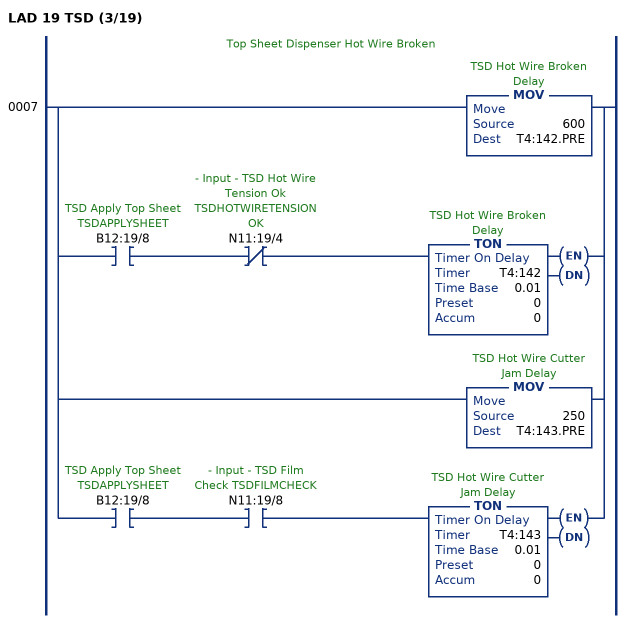
% Rung: 7 %
% Top Sheet Dispenser Hot Wire Broken %
SOR BST MOV 600 T4:142.PRE NXB XIC B12:19/8 XIO N11:19/4 TON T4:142 0.01 0 0 NXB MOV 250 T4:143.PRE NXB XIC B12:19/8 XIC N11:19/8 TON T4:143 0.01 0 0 BND EOR
%   T4:142  "TSD Hot Wire Broken Delay" %
%   B12:19/8  TSDAPPLYSHEET  "TSD Apply Top Sheet" %
%   N11:19/4  TSDHOTWIRETENSIONOK  "- Input - TSD Hot Wire Tension Ok" %
%   T4:143  "TSD Hot Wire Cutter Jam Delay" %
%   N11:19/8  TSDFILMCHECK  "- Input - TSD Film Check" %

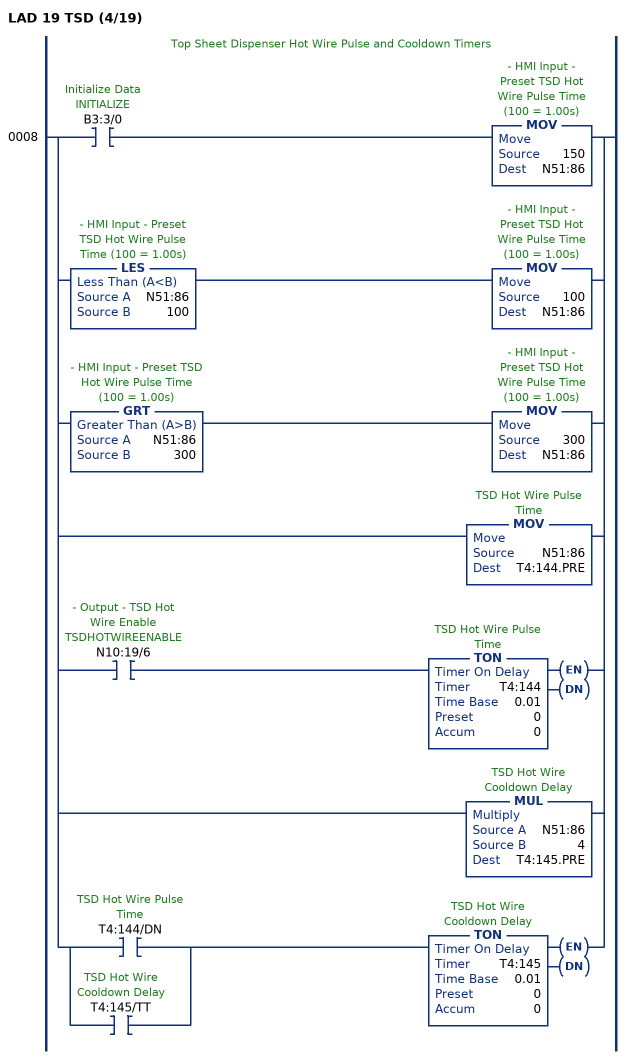
% Rung: 8 %
% Top Sheet Dispenser Hot Wire Pulse and Cooldown Timers %
SOR BST BST XIC B3:3/0 MOV 150 N51:86 NXB LES N51:86 100 MOV 100 N51:86 NXB GRT N51:86 300 MOV 300 N51:86 NXB MOV N51:86 T4:144.PRE BND NXB XIC N10:19/6 TON T4:144 0.01 0 0 NXB MUL N51:86 4 T4:145.PRE NXB BST XIC T4:144/DN NXB XIC T4:145/TT BND TON T4:145 0.01 0 0 BND EOR
%   B3:3/0  INITIALIZE  "Initialize Data" %
%   N51:86  "- HMI Input - Preset TSD Hot Wire Pulse Time (100 = 1.00s)" %
%   T4:144  "TSD Hot Wire Pulse Time" %
%   N10:19/6  TSDHOTWIREENABLE  "- Output - TSD Hot Wire Enable" %
%   T4:145  "TSD Hot Wire Cooldown Delay" %

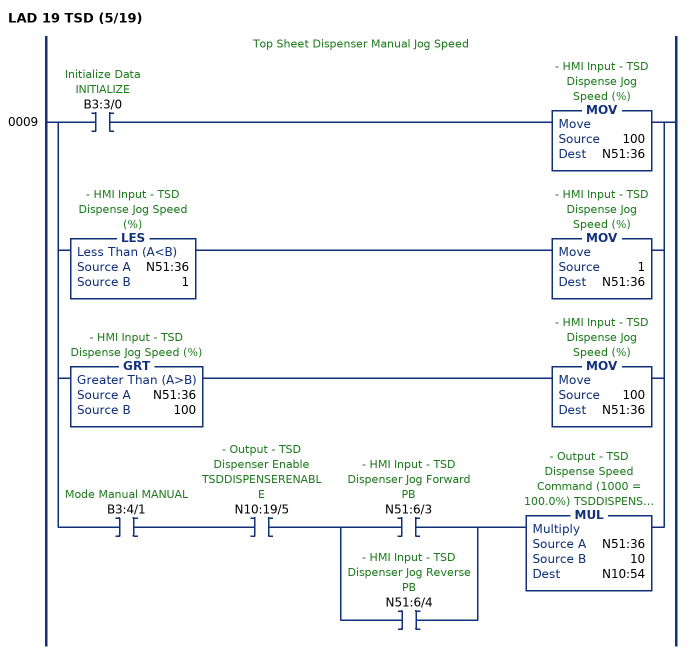
% Rung: 9 %
% Top Sheet Dispenser Manual Jog Speed %
SOR BST XIC B3:3/0 MOV 100 N51:36 NXB LES N51:36 1 MOV 1 N51:36 NXB GRT N51:36 100 MOV 100 N51:36 NXB XIC B3:4/1 XIC N10:19/5 BST XIC N51:6/3 NXB XIC N51:6/4 BND MUL N51:36 10 N10:54 BND EOR
%   B3:3/0  INITIALIZE  "Initialize Data" %
%   N51:36  "- HMI Input - TSD Dispense Jog Speed (%)" %
%   B3:4/1  MANUAL  "Mode Manual" %
%   N10:19/5  TSDDISPENSERENABLE  "- Output - TSD Dispenser Enable" %
%   N51:6/3  "- HMI Input - TSD Dispenser Jog Forward PB" %
%   N51:6/4  "- HMI Input - TSD Dispenser Jog Reverse PB" %
%   N10:54  TSDDISPENSECOMMAND  "- Output - TSD Dispense Speed Command (1000 = 100.0%)" %

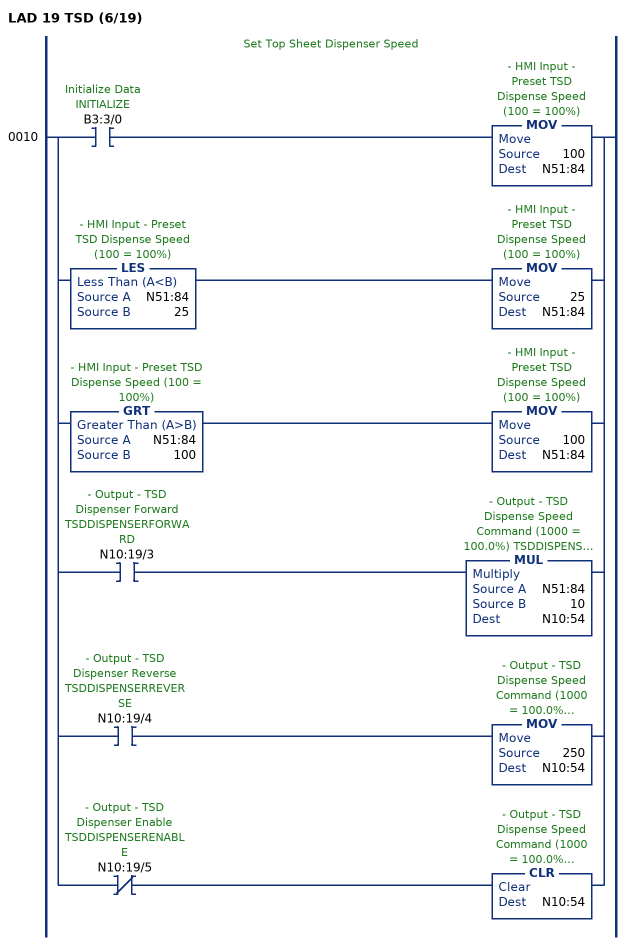
% Rung: 10 %
% Set Top Sheet Dispenser Speed %
SOR BST BST XIC B3:3/0 MOV 100 N51:84 NXB LES N51:84 25 MOV 25 N51:84 NXB GRT N51:84 100 MOV 100 N51:84 BND NXB XIC N10:19/3 MUL N51:84 10 N10:54 NXB XIC N10:19/4 MOV 250 N10:54 NXB XIO N10:19/5 CLR N10:54 BND EOR
%   B3:3/0  INITIALIZE  "Initialize Data" %
%   N51:84  "- HMI Input - Preset TSD Dispense Speed (100 = 100%)" %
%   N10:19/3  TSDDISPENSERFORWARD  "- Output - TSD Dispenser Forward" %
%   N10:54  TSDDISPENSECOMMAND  "- Output - TSD Dispense Speed Command (1000 = 100.0%)" %
%   N10:19/4  TSDDISPENSERREVERSE  "- Output - TSD Dispenser Reverse" %
%   N10:19/5  TSDDISPENSERENABLE  "- Output - TSD Dispenser Enable" %

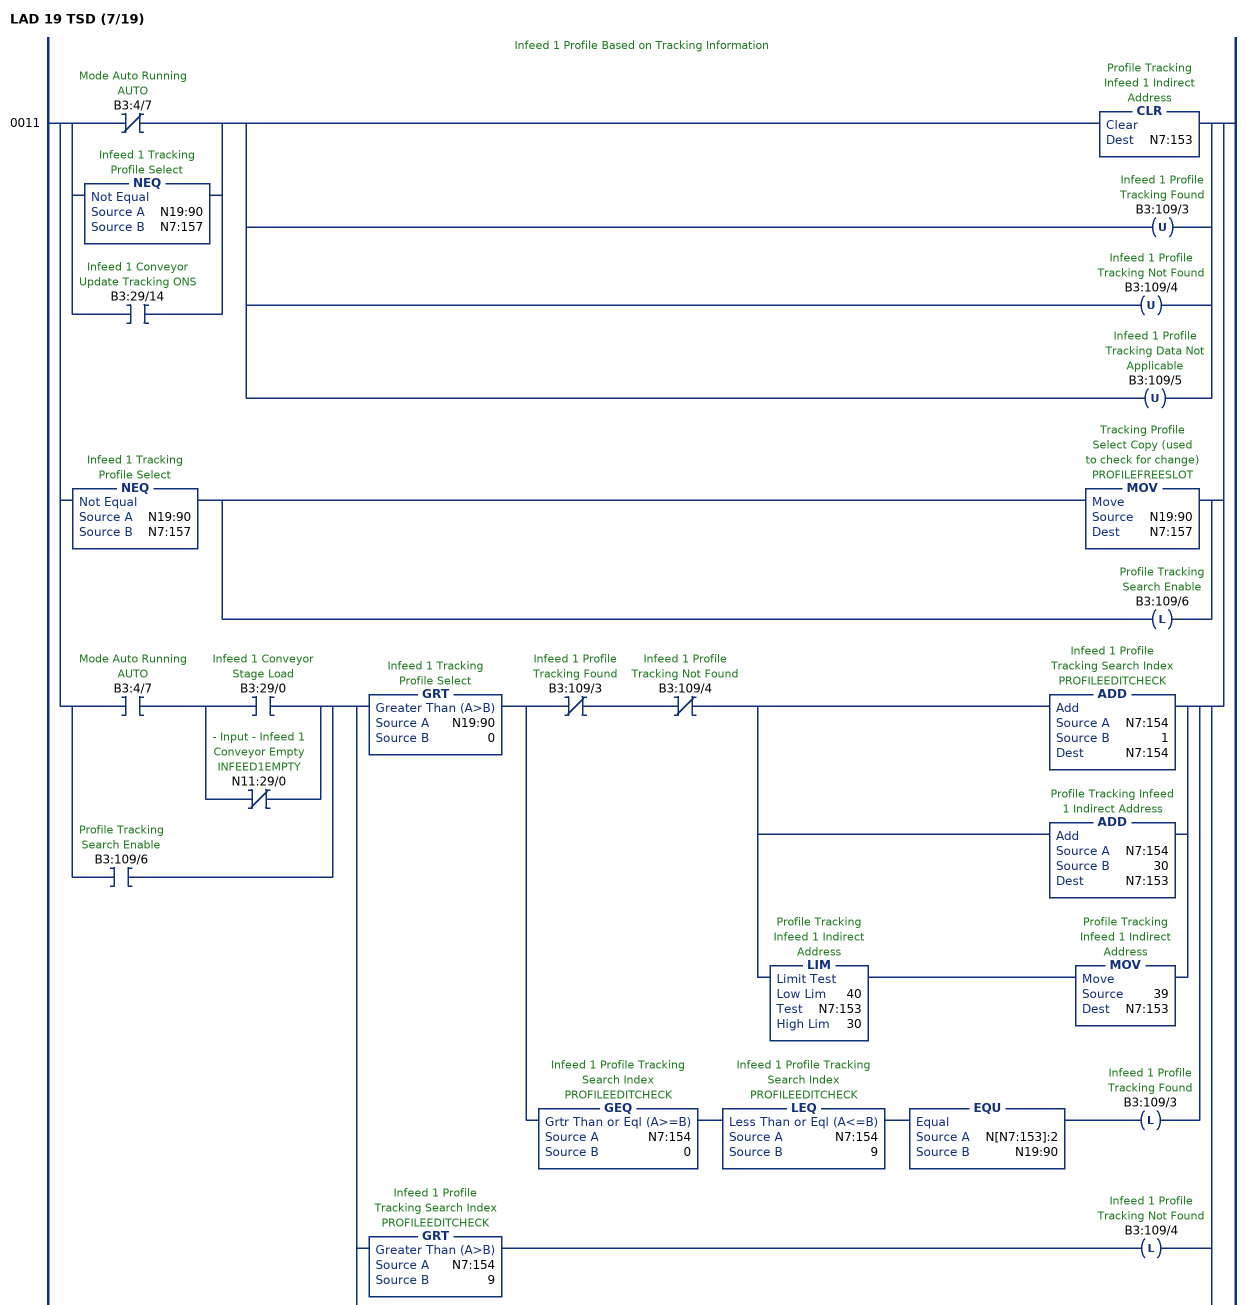

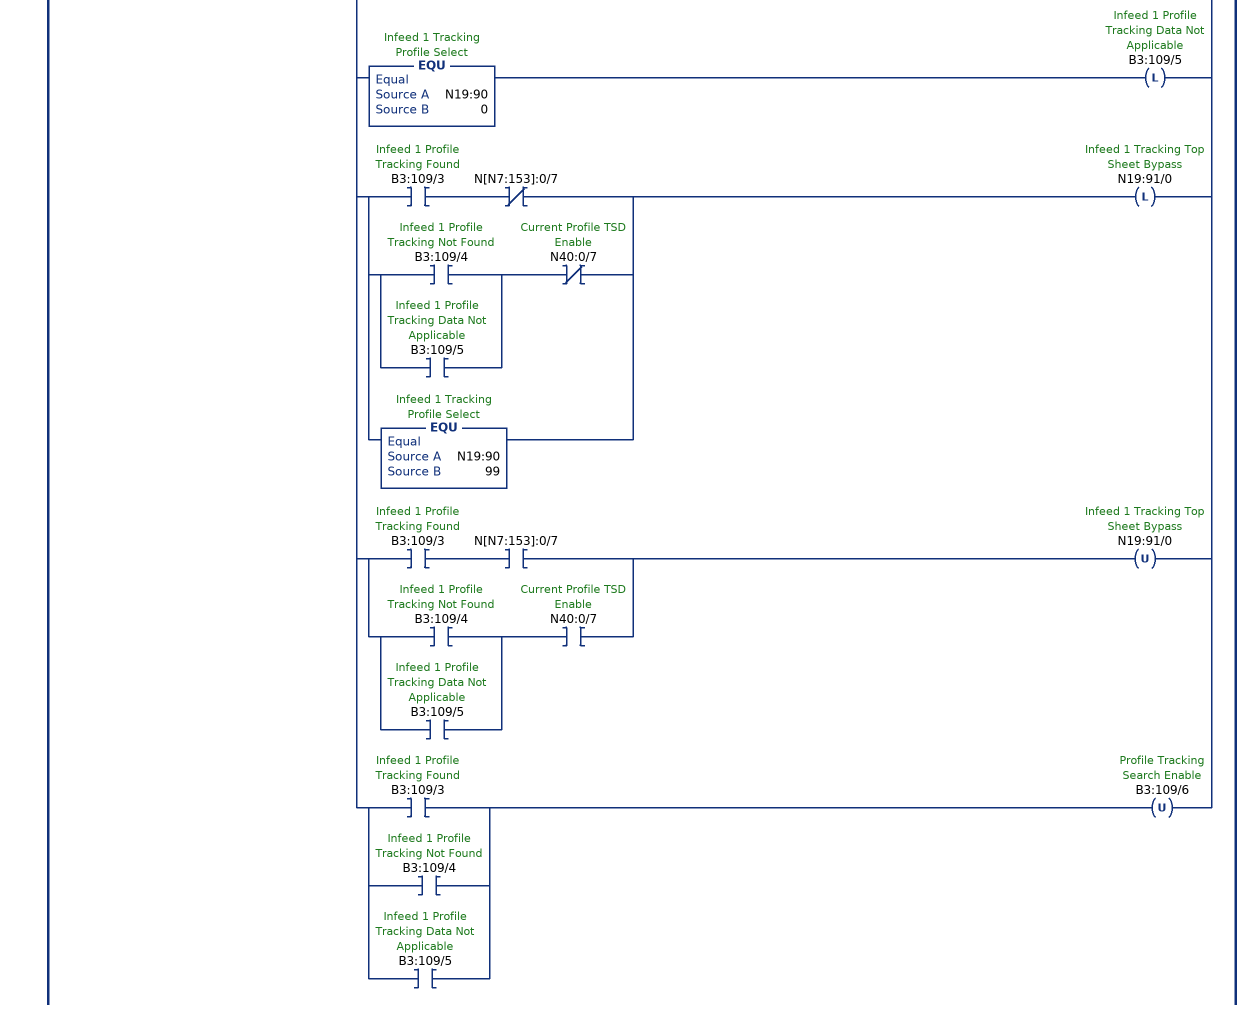
% Rung: 11 %
% Infeed 1 Profile Based on Tracking Information %
SOR BST BST XIO B3:4/7 NXB NEQ N19:90 N7:157 NXB XIC B3:29/14 BND BST CLR N7:153 NXB OTU B3:109/3 NXB OTU B3:109/4 NXB OTU B3:109/5 BND NXB NEQ N19:90 N7:157 BST MOV N19:90 N7:157 NXB OTL B3:109/6 BND NXB BST XIC B3:4/7 BST XIC B3:29/0 NXB XIO N11:29/0 BND NXB XIC B3:109/6 BND BST GRT N19:90 0 BST XIO B3:109/3 XIO B3:109/4 BST ADD N7:154 1 N7:154 NXB ADD N7:154 30 N7:153 NXB LIM 40 N7:153 30 MOV 39 N7:153 BND NXB GEQ N7:154 0 LEQ N7:154 9 EQU N[N7:153]:2 N19:90 OTL B3:109/3 BND NXB GRT N7:154 9 OTL B3:109/4 NXB EQU N19:90 0 OTL B3:109/5 NXB BST XIC B3:109/3 XIO N[N7:153]:0/7 NXB BST XIC B3:109/4 NXB XIC B3:109/5 BND XIO N40:0/7 NXB EQU N19:90 99 BND OTL N19:91/0 NXB BST XIC B3:109/3 XIC N[N7:153]:0/7 NXB BST XIC B3:109/4 NXB XIC B3:109/5 BND XIC N40:0/7 BND OTU N19:91/0 NXB BST XIC B3:109/3 NXB XIC B3:109/4 NXB XIC B3:109/5 BND OTU B3:109/6 BND BND EOR
%   B3:4/7  AUTO  "Mode Auto Running" %
%   N19:90  "Infeed 1 Tracking Profile Select" %
%   N7:157  PROFILEFREESLOT  "Tracking Profile Select Copy (used to check for change)" %
%   B3:29/14  "Infeed 1 Conveyor Update Tracking ONS" %
%   N7:153  "Profile Tracking Infeed 1 Indirect Address" %
%   B3:109/3  "Infeed 1 Profile Tracking Found" %
%   B3:109/4  "Infeed 1 Profile Tracking Not Found" %
%   B3:109/5  "Infeed 1 Profile Tracking Data Not Applicable" %
%   B3:109/6  "Profile Tracking Search Enable" %
%   B3:29/0  "Infeed 1 Conveyor Stage Load" %
%   N11:29/0  INFEED1EMPTY  "- Input - Infeed 1 Conveyor Empty" %
%   N7:154  PROFILEEDITCHECK  "Infeed 1 Profile Tracking Search Index" %
%   N40:0/7  "Current Profile TSD Enable" %
%   N19:91/0  "Infeed 1 Tracking Top Sheet Bypass" %

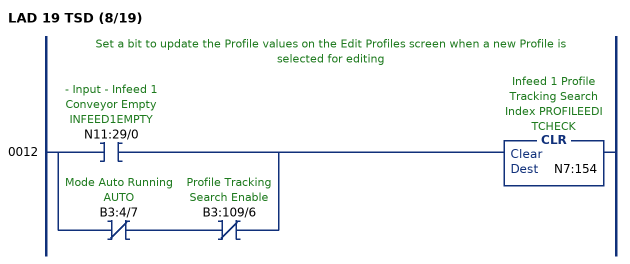
% Rung: 12 %
% Set a bit to update the Profile values on the Edit Profiles screen when a new Profile is selected for editing %
SOR BST XIC N11:29/0 NXB XIO B3:4/7 XIO B3:109/6 BND CLR N7:154 EOR
%   N11:29/0  INFEED1EMPTY  "- Input - Infeed 1 Conveyor Empty" %
%   B3:4/7  AUTO  "Mode Auto Running" %
%   B3:109/6  "Profile Tracking Search Enable" %
%   N7:154  PROFILEEDITCHECK  "Infeed 1 Profile Tracking Search Index" %

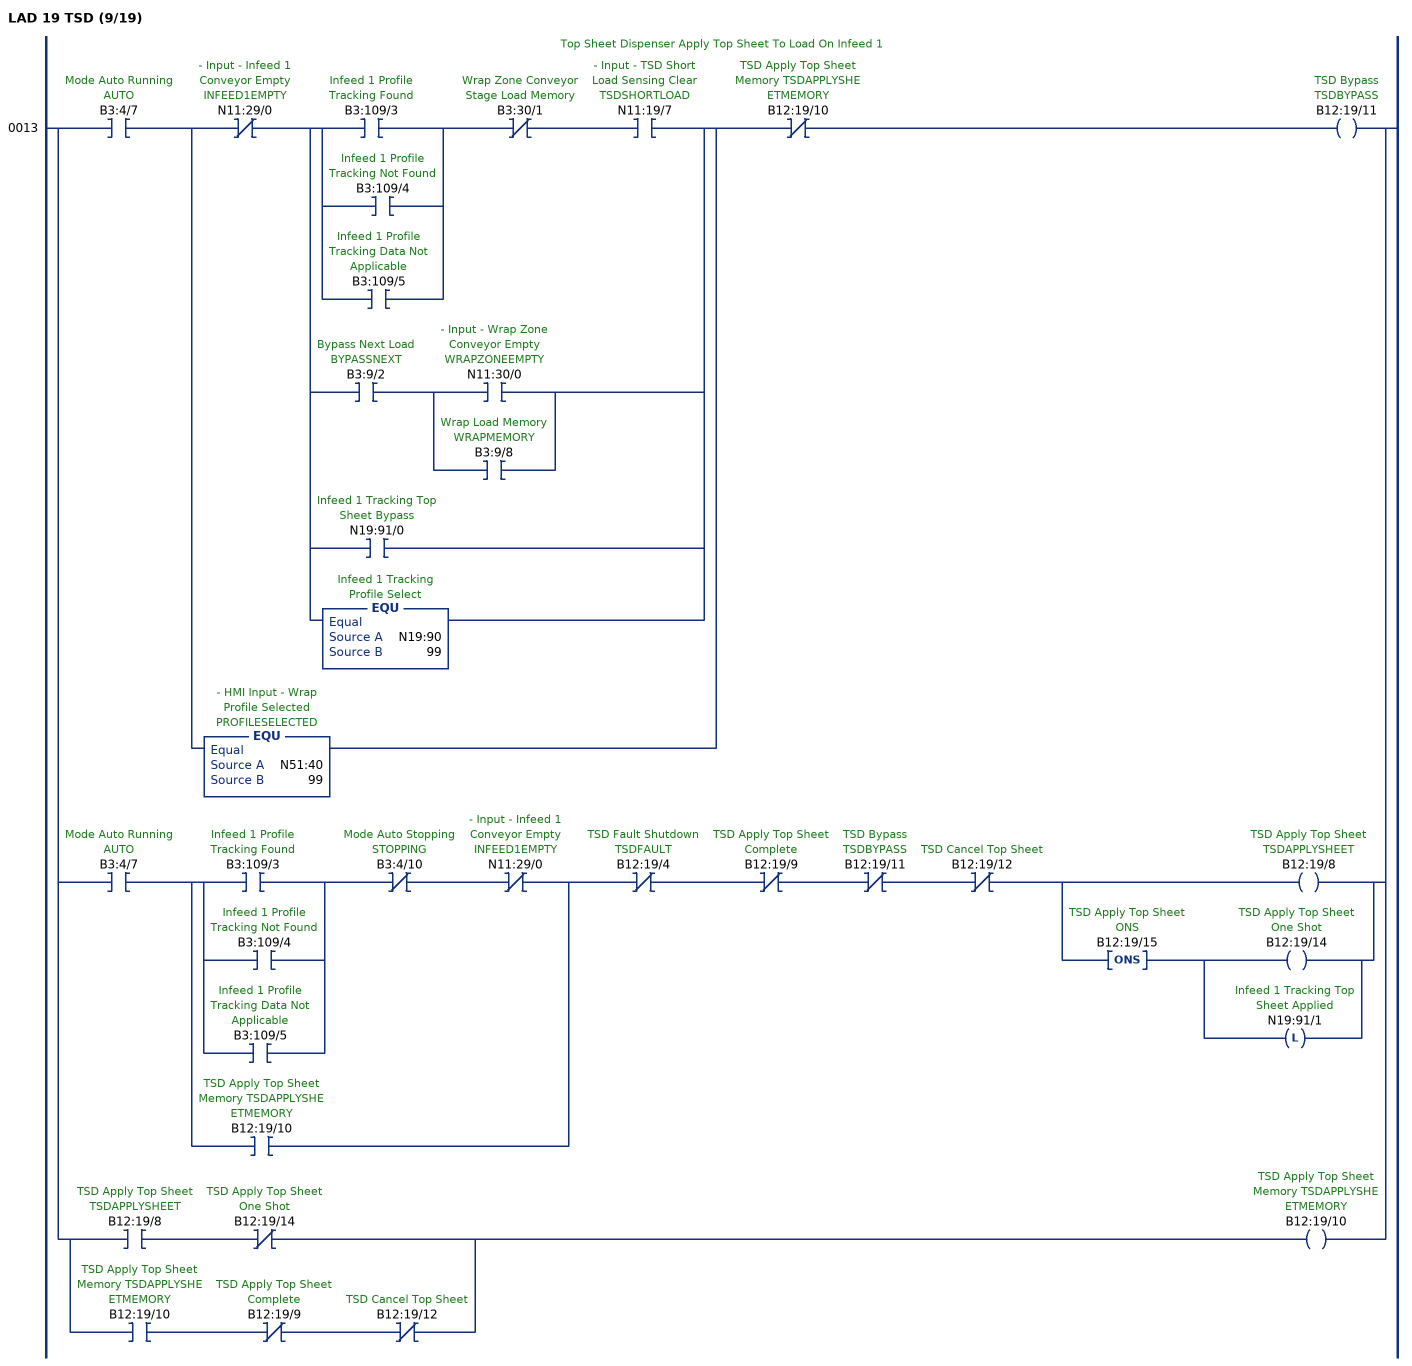
% Rung: 13 %
% Top Sheet Dispenser Apply Top Sheet To Load On Infeed 1 %
SOR BST XIC B3:4/7 BST XIO N11:29/0 BST BST XIC B3:109/3 NXB XIC B3:109/4 NXB XIC B3:109/5 BND XIO B3:30/1 XIC N11:19/7 NXB XIC B3:9/2 BST XIC N11:30/0 NXB XIC B3:9/8 BND NXB XIC N19:91/0 NXB EQU N19:90 99 BND NXB EQU N51:40 99 BND XIO B12:19/10 OTE B12:19/11 NXB XIC B3:4/7 BST BST XIC B3:109/3 NXB XIC B3:109/4 NXB XIC B3:109/5 BND XIO B3:4/10 XIO N11:29/0 NXB XIC B12:19/10 BND XIO B12:19/4 XIO B12:19/9 XIO B12:19/11 XIO B12:19/12 BST OTE B12:19/8 NXB ONS B12:19/15 BST OTE B12:19/14 NXB OTL N19:91/1 BND BND NXB BST XIC B12:19/8 XIO B12:19/14 NXB XIC B12:19/10 XIO B12:19/9 XIO B12:19/12 BND OTE B12:19/10 BND EOR
%   B3:4/7  AUTO  "Mode Auto Running" %
%   N11:29/0  INFEED1EMPTY  "- Input - Infeed 1 Conveyor Empty" %
%   B3:109/3  "Infeed 1 Profile Tracking Found" %
%   B3:109/4  "Infeed 1 Profile Tracking Not Found" %
%   B3:109/5  "Infeed 1 Profile Tracking Data Not Applicable" %
%   B3:30/1  "Wrap Zone Conveyor Stage Load Memory" %
%   N11:19/7  TSDSHORTLOAD  "- Input - TSD Short Load Sensing Clear" %
%   B3:9/2  BYPASSNEXT  "Bypass Next Load" %
%   N11:30/0  WRAPZONEEMPTY  "- Input - Wrap Zone Conveyor Empty" %
%   B3:9/8  WRAPMEMORY  "Wrap Load Memory" %
%   N19:91/0  "Infeed 1 Tracking Top Sheet Bypass" %
%   N19:90  "Infeed 1 Tracking Profile Select" %
%   N51:40  PROFILESELECTED  "- HMI Input - Wrap Profile Selected" %
%   B12:19/10  TSDAPPLYSHEETMEMORY  "TSD Apply Top Sheet Memory" %
%   B12:19/11  TSDBYPASS  "TSD Bypass" %
%   B3:4/10  STOPPING  "Mode Auto Stopping" %
%   B12:19/4  TSDFAULT  "TSD Fault Shutdown" %
%   B12:19/9  "TSD Apply Top Sheet Complete" %
%   B12:19/12  "TSD Cancel Top Sheet" %
%   B12:19/8  TSDAPPLYSHEET  "TSD Apply Top Sheet" %
%   B12:19/15  "TSD Apply Top Sheet ONS" %
%   B12:19/14  "TSD Apply Top Sheet One Shot" %
%   N19:91/1  "Infeed 1 Tracking Top Sheet Applied" %

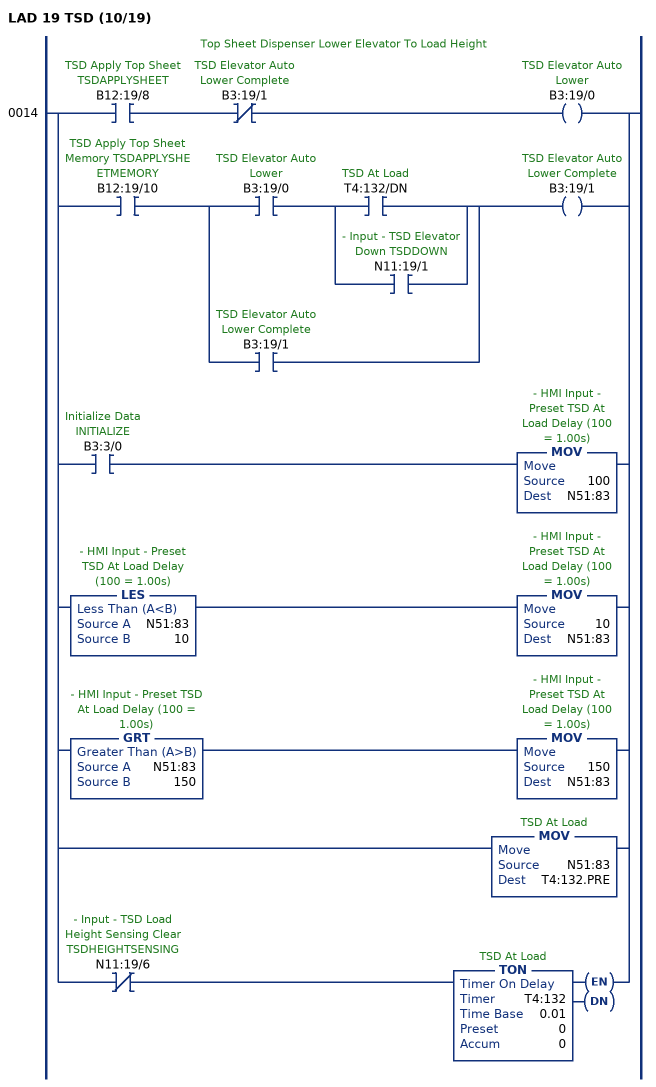
% Rung: 14 %
% Top Sheet Dispenser Lower Elevator To Load Height %
SOR BST XIC B12:19/8 XIO B3:19/1 OTE B3:19/0 NXB XIC B12:19/10 BST XIC B3:19/0 BST XIC T4:132/DN NXB XIC N11:19/1 BND NXB XIC B3:19/1 BND OTE B3:19/1 NXB BST XIC B3:3/0 MOV 100 N51:83 NXB LES N51:83 10 MOV 10 N51:83 NXB GRT N51:83 150 MOV 150 N51:83 NXB MOV N51:83 T4:132.PRE BND NXB XIO N11:19/6 TON T4:132 0.01 0 0 BND EOR
%   B12:19/8  TSDAPPLYSHEET  "TSD Apply Top Sheet" %
%   B3:19/1  "TSD Elevator Auto Lower Complete" %
%   B3:19/0  "TSD Elevator Auto Lower" %
%   B12:19/10  TSDAPPLYSHEETMEMORY  "TSD Apply Top Sheet Memory" %
%   T4:132  "TSD At Load" %
%   N11:19/1  TSDDOWN  "- Input - TSD Elevator Down" %
%   B3:3/0  INITIALIZE  "Initialize Data" %
%   N51:83  "- HMI Input - Preset TSD At Load Delay (100 = 1.00s)" %
%   N11:19/6  TSDHEIGHTSENSING  "- Input - TSD Load Height Sensing Clear" %

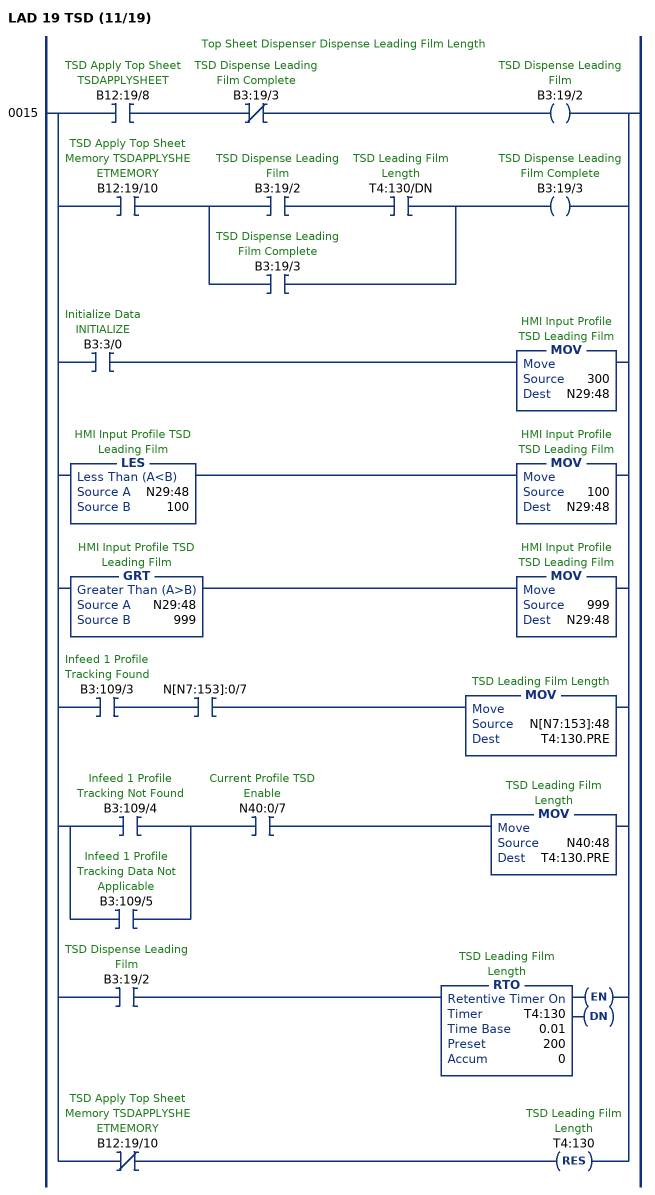
% Rung: 15 %
% Top Sheet Dispenser Dispense Leading Film Length %
SOR BST XIC B12:19/8 XIO B3:19/3 OTE B3:19/2 NXB XIC B12:19/10 BST XIC B3:19/2 XIC T4:130/DN NXB XIC B3:19/3 BND OTE B3:19/3 NXB BST XIC B3:3/0 MOV 300 N29:48 NXB LES N29:48 100 MOV 100 N29:48 NXB GRT N29:48 999 MOV 999 N29:48 NXB XIC B3:109/3 XIC N[N7:153]:0/7 MOV N[N7:153]:48 T4:130.PRE NXB BST XIC B3:109/4 NXB XIC B3:109/5 BND XIC N40:0/7 MOV N40:48 T4:130.PRE BND NXB XIC B3:19/2 RTO T4:130 0.01 200 0 NXB XIO B12:19/10 RES T4:130 BND EOR
%   B12:19/8  TSDAPPLYSHEET  "TSD Apply Top Sheet" %
%   B3:19/3  "TSD Dispense Leading Film Complete" %
%   B3:19/2  "TSD Dispense Leading Film" %
%   B12:19/10  TSDAPPLYSHEETMEMORY  "TSD Apply Top Sheet Memory" %
%   T4:130  "TSD Leading Film Length" %
%   B3:3/0  INITIALIZE  "Initialize Data" %
%   N29:48  "HMI Input Profile TSD Leading Film" %
%   B3:109/3  "Infeed 1 Profile Tracking Found" %
%   N7:153  "Profile Tracking Infeed 1 Indirect Address" %
%   B3:109/4  "Infeed 1 Profile Tracking Not Found" %
%   B3:109/5  "Infeed 1 Profile Tracking Data Not Applicable" %
%   N40:0/7  "Current Profile TSD Enable" %
%   N40:48  "Current Profile TSD Leading Film" %

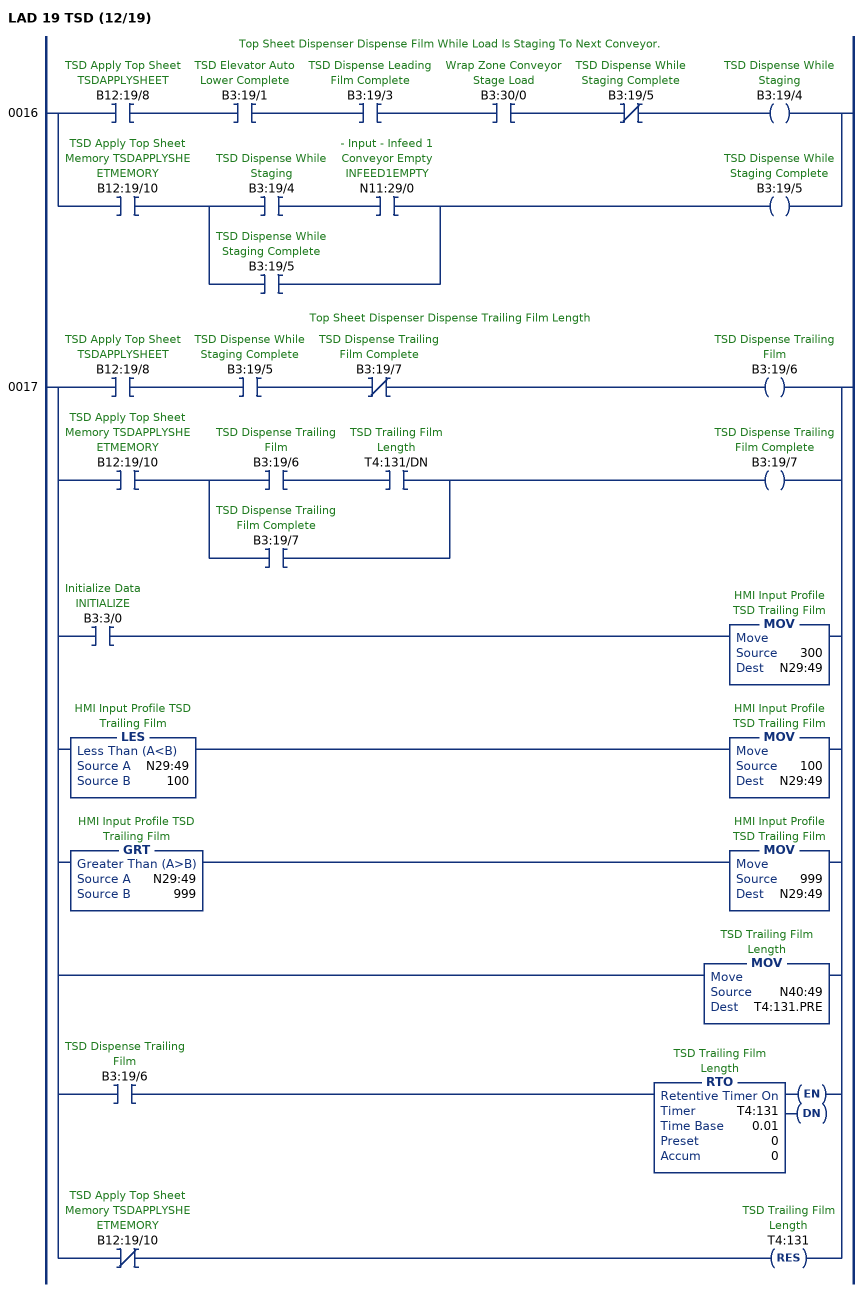
% Rung: 16 %
% Top Sheet Dispenser Dispense Film While Load Is Staging To Next Conveyor. %
SOR BST XIC B12:19/8 XIC B3:19/1 XIC B3:19/3 XIC B3:30/0 XIO B3:19/5 OTE B3:19/4 NXB XIC B12:19/10 BST XIC B3:19/4 XIC N11:29/0 NXB XIC B3:19/5 BND OTE B3:19/5 BND EOR
%   B12:19/8  TSDAPPLYSHEET  "TSD Apply Top Sheet" %
%   B3:19/1  "TSD Elevator Auto Lower Complete" %
%   B3:19/3  "TSD Dispense Leading Film Complete" %
%   B3:30/0  "Wrap Zone Conveyor Stage Load" %
%   B3:19/5  "TSD Dispense While Staging Complete" %
%   B3:19/4  "TSD Dispense While Staging" %
%   B12:19/10  TSDAPPLYSHEETMEMORY  "TSD Apply Top Sheet Memory" %
%   N11:29/0  INFEED1EMPTY  "- Input - Infeed 1 Conveyor Empty" %
% Rung: 17 %
% Top Sheet Dispenser Dispense Trailing Film Length %
SOR BST XIC B12:19/8 XIC B3:19/5 XIO B3:19/7 OTE B3:19/6 NXB XIC B12:19/10 BST XIC B3:19/6 XIC T4:131/DN NXB XIC B3:19/7 BND OTE B3:19/7 NXB BST XIC B3:3/0 MOV 300 N29:49 NXB LES N29:49 100 MOV 100 N29:49 NXB GRT N29:49 999 MOV 999 N29:49 NXB MOV N40:49 T4:131.PRE BND NXB XIC B3:19/6 RTO T4:131 0.01 0 0 NXB XIO B12:19/10 RES T4:131 BND EOR
%   B12:19/8  TSDAPPLYSHEET  "TSD Apply Top Sheet" %
%   B3:19/5  "TSD Dispense While Staging Complete" %
%   B3:19/7  "TSD Dispense Trailing Film Complete" %
%   B3:19/6  "TSD Dispense Trailing Film" %
%   B12:19/10  TSDAPPLYSHEETMEMORY  "TSD Apply Top Sheet Memory" %
%   T4:131  "TSD Trailing Film Length" %
%   B3:3/0  INITIALIZE  "Initialize Data" %
%   N29:49  "HMI Input Profile TSD Trailing Film" %
%   N40:49  "Current Profile TSD Trailing Film" %

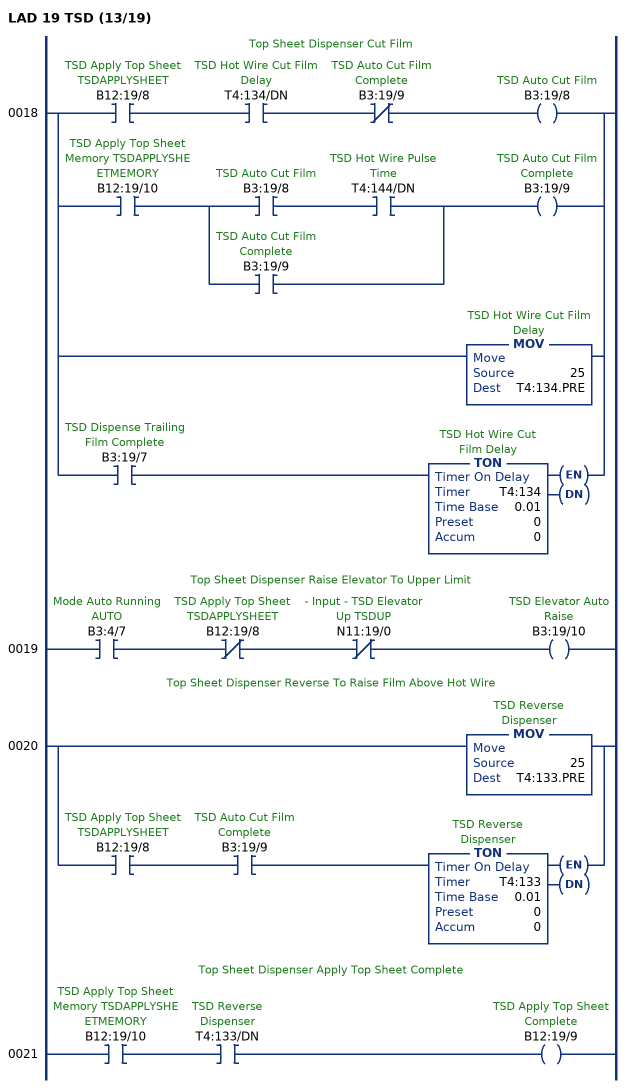
% Rung: 18 %
% Top Sheet Dispenser Cut Film %
SOR BST XIC B12:19/8 XIC T4:134/DN XIO B3:19/9 OTE B3:19/8 NXB XIC B12:19/10 BST XIC B3:19/8 XIC T4:144/DN NXB XIC B3:19/9 BND OTE B3:19/9 NXB MOV 25 T4:134.PRE NXB XIC B3:19/7 TON T4:134 0.01 0 0 BND EOR
%   B12:19/8  TSDAPPLYSHEET  "TSD Apply Top Sheet" %
%   T4:134  "TSD Hot Wire Cut Film Delay" %
%   B3:19/9  "TSD Auto Cut Film Complete" %
%   B3:19/8  "TSD Auto Cut Film" %
%   B12:19/10  TSDAPPLYSHEETMEMORY  "TSD Apply Top Sheet Memory" %
%   T4:144  "TSD Hot Wire Pulse Time" %
%   B3:19/7  "TSD Dispense Trailing Film Complete" %
% Rung: 19 %
% Top Sheet Dispenser Raise Elevator To Upper Limit %
SOR XIC B3:4/7 XIO B12:19/8 XIO N11:19/0 OTE B3:19/10 EOR
%   B3:4/7  AUTO  "Mode Auto Running" %
%   B12:19/8  TSDAPPLYSHEET  "TSD Apply Top Sheet" %
%   N11:19/0  TSDUP  "- Input - TSD Elevator Up" %
%   B3:19/10  "TSD Elevator Auto Raise" %
% Rung: 20 %
% Top Sheet Dispenser Reverse To Raise Film Above Hot Wire %
SOR BST MOV 25 T4:133.PRE NXB XIC B12:19/8 XIC B3:19/9 TON T4:133 0.01 0 0 BND EOR
%   T4:133  "TSD Reverse Dispenser" %
%   B12:19/8  TSDAPPLYSHEET  "TSD Apply Top Sheet" %
%   B3:19/9  "TSD Auto Cut Film Complete" %
% Rung: 21 %
% Top Sheet Dispenser Apply Top Sheet Complete %
SOR XIC B12:19/10 XIC T4:133/DN OTE B12:19/9 EOR
%   B12:19/10  TSDAPPLYSHEETMEMORY  "TSD Apply Top Sheet Memory" %
%   T4:133  "TSD Reverse Dispenser" %
%   B12:19/9  "TSD Apply Top Sheet Complete" %

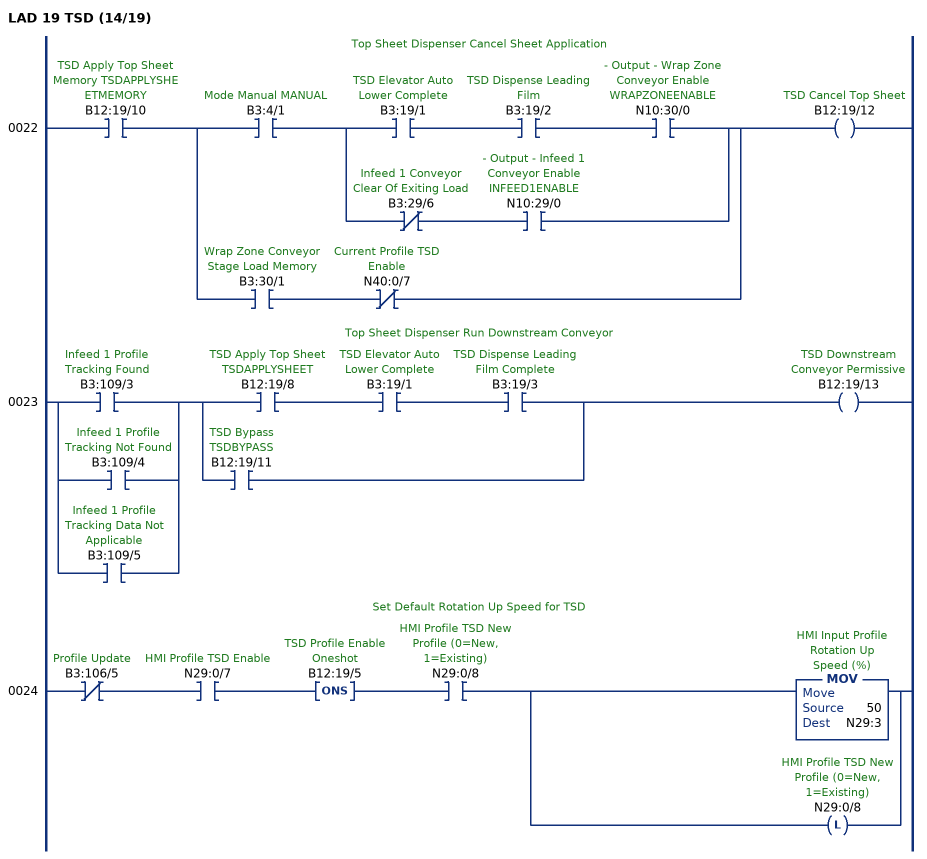
% Rung: 22 %
% Top Sheet Dispenser Cancel Sheet Application %
SOR XIC B12:19/10 BST XIC B3:4/1 BST XIC B3:19/1 XIC B3:19/2 XIC N10:30/0 NXB XIO B3:29/6 XIC N10:29/0 BND NXB XIC B3:30/1 XIO N40:0/7 BND OTE B12:19/12 EOR
%   B12:19/10  TSDAPPLYSHEETMEMORY  "TSD Apply Top Sheet Memory" %
%   B3:4/1  MANUAL  "Mode Manual" %
%   B3:19/1  "TSD Elevator Auto Lower Complete" %
%   B3:19/2  "TSD Dispense Leading Film" %
%   N10:30/0  WRAPZONEENABLE  "- Output - Wrap Zone Conveyor Enable" %
%   B3:29/6  "Infeed 1 Conveyor Clear Of Exiting Load" %
%   N10:29/0  INFEED1ENABLE  "- Output - Infeed 1 Conveyor Enable" %
%   B3:30/1  "Wrap Zone Conveyor Stage Load Memory" %
%   N40:0/7  "Current Profile TSD Enable" %
%   B12:19/12  "TSD Cancel Top Sheet" %
% Rung: 23 %
% Top Sheet Dispenser Run Downstream Conveyor %
SOR BST XIC B3:109/3 NXB XIC B3:109/4 NXB XIC B3:109/5 BND BST XIC B12:19/8 XIC B3:19/1 XIC B3:19/3 NXB XIC B12:19/11 BND OTE B12:19/13 EOR
%   B3:109/3  "Infeed 1 Profile Tracking Found" %
%   B3:109/4  "Infeed 1 Profile Tracking Not Found" %
%   B3:109/5  "Infeed 1 Profile Tracking Data Not Applicable" %
%   B12:19/8  TSDAPPLYSHEET  "TSD Apply Top Sheet" %
%   B3:19/1  "TSD Elevator Auto Lower Complete" %
%   B3:19/3  "TSD Dispense Leading Film Complete" %
%   B12:19/11  TSDBYPASS  "TSD Bypass" %
%   B12:19/13  "TSD Downstream Conveyor Permissive" %
% Rung: 24 %
% Set Default Rotation Up Speed for TSD %
SOR XIO B3:106/5 XIC N29:0/7 ONS B12:19/5 XIC N29:0/8 BST MOV 50 N29:3 NXB OTL N29:0/8 BND EOR
%   B3:106/5  "Profile Update" %
%   N29:0/7  "HMI Profile TSD Enable" %
%   B12:19/5  "TSD Profile Enable Oneshot" %
%   N29:0/8  "HMI Profile TSD New Profile (0=New, 1=Existing)" %
%   N29:3  "HMI Input Profile Rotation Up Speed (%)" %

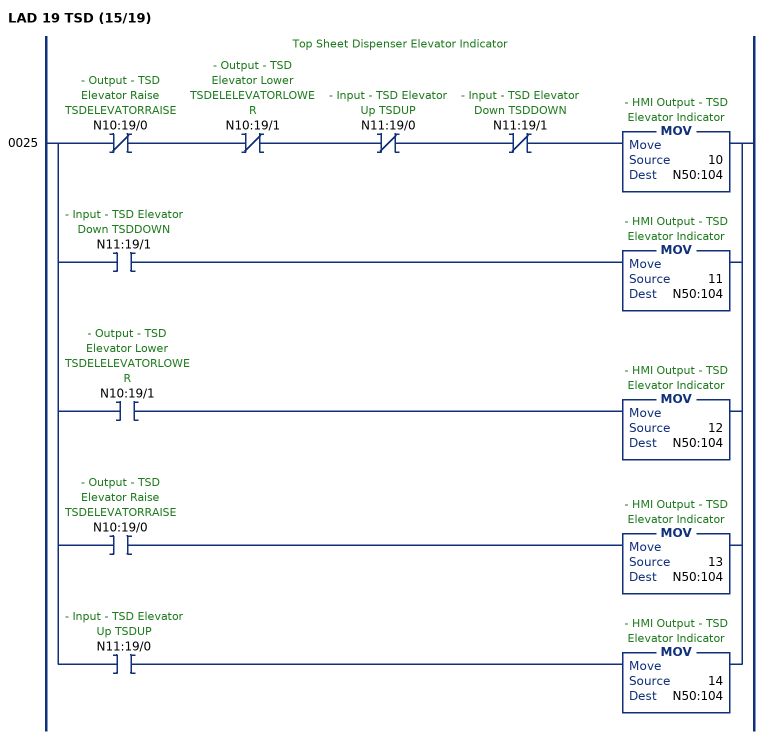
% Rung: 25 %
% Top Sheet Dispenser Elevator Indicator %
SOR BST XIO N10:19/0 XIO N10:19/1 XIO N11:19/0 XIO N11:19/1 MOV 10 N50:104 NXB XIC N11:19/1 MOV 11 N50:104 NXB XIC N10:19/1 MOV 12 N50:104 NXB XIC N10:19/0 MOV 13 N50:104 NXB XIC N11:19/0 MOV 14 N50:104 BND EOR
%   N10:19/0  TSDELEVATORRAISE  "- Output - TSD Elevator Raise" %
%   N10:19/1  TSDELELEVATORLOWER  "- Output - TSD Elevator Lower" %
%   N11:19/0  TSDUP  "- Input - TSD Elevator Up" %
%   N11:19/1  TSDDOWN  "- Input - TSD Elevator Down" %
%   N50:104  "- HMI Output - TSD Elevator Indicator" %

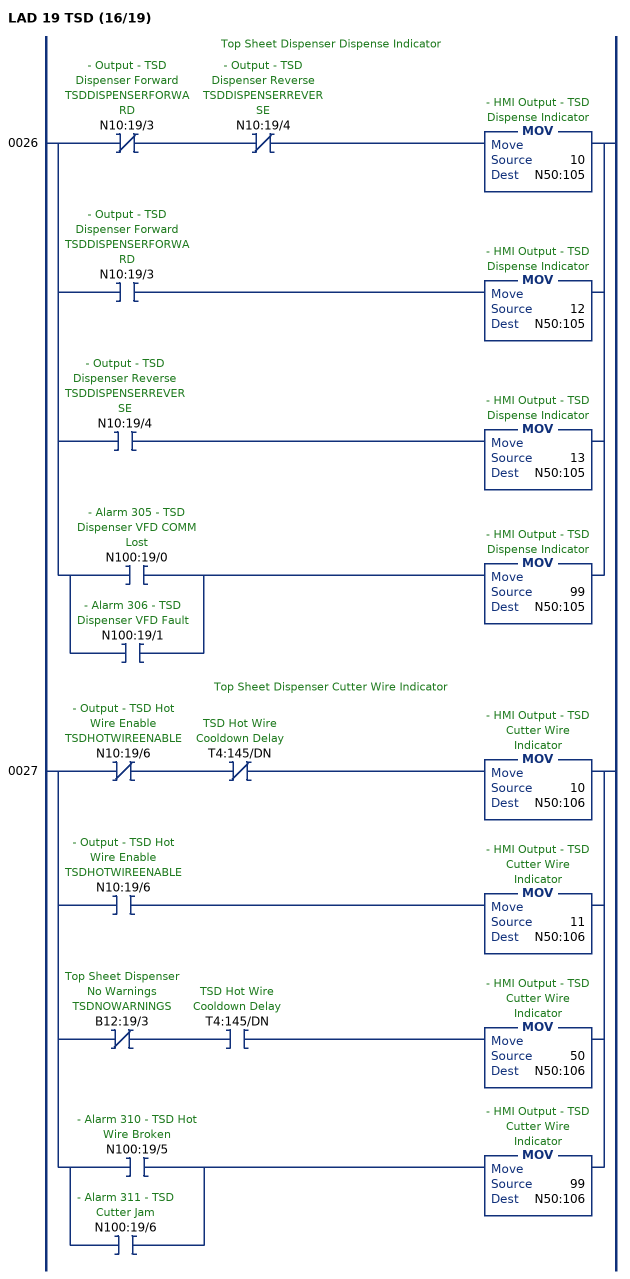
% Rung: 26 %
% Top Sheet Dispenser Dispense Indicator %
SOR BST XIO N10:19/3 XIO N10:19/4 MOV 10 N50:105 NXB XIC N10:19/3 MOV 12 N50:105 NXB XIC N10:19/4 MOV 13 N50:105 NXB BST XIC N100:19/0 NXB XIC N100:19/1 BND MOV 99 N50:105 BND EOR
%   N10:19/3  TSDDISPENSERFORWARD  "- Output - TSD Dispenser Forward" %
%   N10:19/4  TSDDISPENSERREVERSE  "- Output - TSD Dispenser Reverse" %
%   N50:105  "- HMI Output - TSD Dispense Indicator" %
%   N100:19/0  "- Alarm 305 - TSD Dispenser VFD COMM Lost" %
%   N100:19/1  "- Alarm 306 - TSD Dispenser VFD Fault" %
% Rung: 27 %
% Top Sheet Dispenser Cutter Wire Indicator %
SOR BST XIO N10:19/6 XIO T4:145/DN MOV 10 N50:106 NXB XIC N10:19/6 MOV 11 N50:106 NXB XIO B12:19/3 XIC T4:145/DN MOV 50 N50:106 NXB BST XIC N100:19/5 NXB XIC N100:19/6 BND MOV 99 N50:106 BND EOR
%   N10:19/6  TSDHOTWIREENABLE  "- Output - TSD Hot Wire Enable" %
%   T4:145  "TSD Hot Wire Cooldown Delay" %
%   N50:106  "- HMI Output - TSD Cutter Wire Indicator" %
%   B12:19/3  TSDNOWARNINGS  "Top Sheet Dispenser No Warnings" %
%   N100:19/5  "- Alarm 310 - TSD Hot Wire Broken" %
%   N100:19/6  "- Alarm 311 - TSD Cutter Jam" %

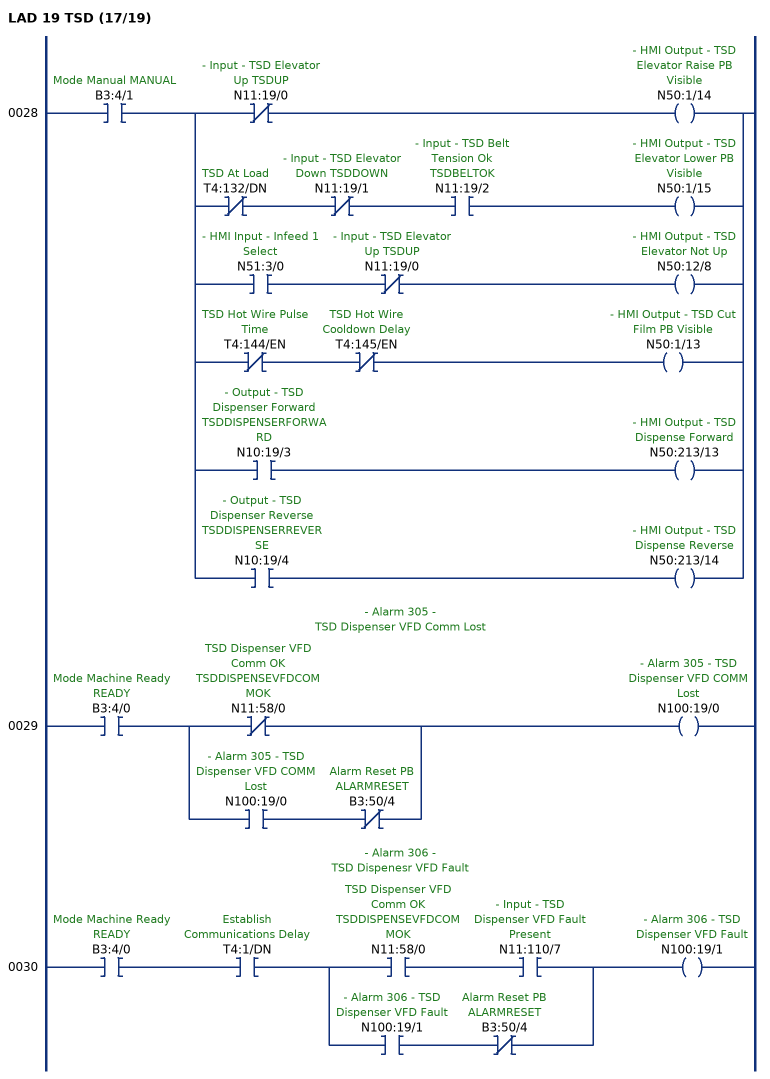
% Rung: 28 %
SOR XIC B3:4/1 BST XIO N11:19/0 OTE N50:1/14 NXB XIO T4:132/DN XIO N11:19/1 XIC N11:19/2 OTE N50:1/15 NXB XIC N51:3/0 XIO N11:19/0 OTE N50:12/8 NXB XIO T4:144/EN XIO T4:145/EN OTE N50:1/13 NXB XIC N10:19/3 OTE N50:213/13 NXB XIC N10:19/4 OTE N50:213/14 BND EOR
%   B3:4/1  MANUAL  "Mode Manual" %
%   N11:19/0  TSDUP  "- Input - TSD Elevator Up" %
%   N50:1/14  "- HMI Output - TSD Elevator Raise PB Visible" %
%   T4:132  "TSD At Load" %
%   N11:19/1  TSDDOWN  "- Input - TSD Elevator Down" %
%   N11:19/2  TSDBELTOK  "- Input - TSD Belt Tension Ok" %
%   N50:1/15  "- HMI Output - TSD Elevator Lower PB Visible" %
%   N51:3/0  "- HMI Input - Infeed 1 Select" %
%   N50:12/8  "- HMI Output - TSD Elevator Not Up" %
%   T4:144  "TSD Hot Wire Pulse Time" %
%   T4:145  "TSD Hot Wire Cooldown Delay" %
%   N50:1/13  "- HMI Output - TSD Cut Film PB Visible" %
%   N10:19/3  TSDDISPENSERFORWARD  "- Output - TSD Dispenser Forward" %
%   N50:213/13  "- HMI Output - TSD Dispense Forward" %
%   N10:19/4  TSDDISPENSERREVERSE  "- Output - TSD Dispenser Reverse" %
%   N50:213/14  "- HMI Output - TSD Dispense Reverse" %
% Rung: 29 %
% - Alarm 305 -
% 
% TSD Dispenser VFD Comm Lost %
SOR XIC B3:4/0 BST XIO N11:58/0 NXB XIC N100:19/0 XIO B3:50/4 BND OTE N100:19/0 EOR
%   B3:4/0  READY  "Mode Machine Ready" %
%   N11:58/0  TSDDISPENSEVFDCOMMOK  "TSD Dispenser VFD Comm OK" %
%   N100:19/0  "- Alarm 305 - TSD Dispenser VFD COMM Lost" %
%   B3:50/4  ALARMRESET  "Alarm Reset PB" %
% Rung: 30 %
% - Alarm 306 -
% 
% TSD Dispenesr VFD Fault %
SOR XIC B3:4/0 XIC T4:1/DN BST XIC N11:58/0 XIC N11:110/7 NXB XIC N100:19/1 XIO B3:50/4 BND OTE N100:19/1 EOR
%   B3:4/0  READY  "Mode Machine Ready" %
%   T4:1  "Establish Communications Delay" %
%   N11:58/0  TSDDISPENSEVFDCOMMOK  "TSD Dispenser VFD Comm OK" %
%   N11:110/7  "- Input - TSD Dispenser VFD Fault Present" %
%   N100:19/1  "- Alarm 306 - TSD Dispenser VFD Fault" %
%   B3:50/4  ALARMRESET  "Alarm Reset PB" %

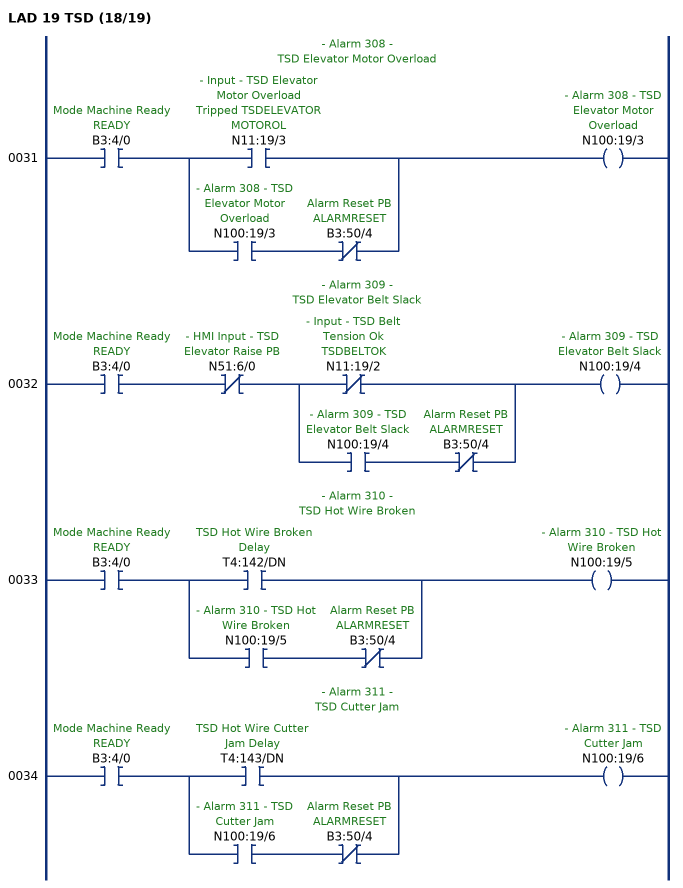
% Rung: 31 %
% - Alarm 308 -
% 
% TSD Elevator Motor Overload %
SOR XIC B3:4/0 BST XIC N11:19/3 NXB XIC N100:19/3 XIO B3:50/4 BND OTE N100:19/3 EOR
%   B3:4/0  READY  "Mode Machine Ready" %
%   N11:19/3  TSDELEVATORMOTOROL  "- Input - TSD Elevator Motor Overload Tripped" %
%   N100:19/3  "- Alarm 308 - TSD Elevator Motor Overload" %
%   B3:50/4  ALARMRESET  "Alarm Reset PB" %
% Rung: 32 %
% - Alarm 309 -
% 
% TSD Elevator Belt Slack %
SOR XIC B3:4/0 XIO N51:6/0 BST XIO N11:19/2 NXB XIC N100:19/4 XIO B3:50/4 BND OTE N100:19/4 EOR
%   B3:4/0  READY  "Mode Machine Ready" %
%   N51:6/0  "- HMI Input - TSD Elevator Raise PB" %
%   N11:19/2  TSDBELTOK  "- Input - TSD Belt Tension Ok" %
%   N100:19/4  "- Alarm 309 - TSD Elevator Belt Slack" %
%   B3:50/4  ALARMRESET  "Alarm Reset PB" %
% Rung: 33 %
% - Alarm 310 -
% 
% TSD Hot Wire Broken %
SOR XIC B3:4/0 BST XIC T4:142/DN NXB XIC N100:19/5 XIO B3:50/4 BND OTE N100:19/5 EOR
%   B3:4/0  READY  "Mode Machine Ready" %
%   T4:142  "TSD Hot Wire Broken Delay" %
%   N100:19/5  "- Alarm 310 - TSD Hot Wire Broken" %
%   B3:50/4  ALARMRESET  "Alarm Reset PB" %
% Rung: 34 %
% - Alarm 311 -
% 
% TSD Cutter Jam %
SOR XIC B3:4/0 BST XIC T4:143/DN NXB XIC N100:19/6 XIO B3:50/4 BND OTE N100:19/6 EOR
%   B3:4/0  READY  "Mode Machine Ready" %
%   T4:143  "TSD Hot Wire Cutter Jam Delay" %
%   N100:19/6  "- Alarm 311 - TSD Cutter Jam" %
%   B3:50/4  ALARMRESET  "Alarm Reset PB" %

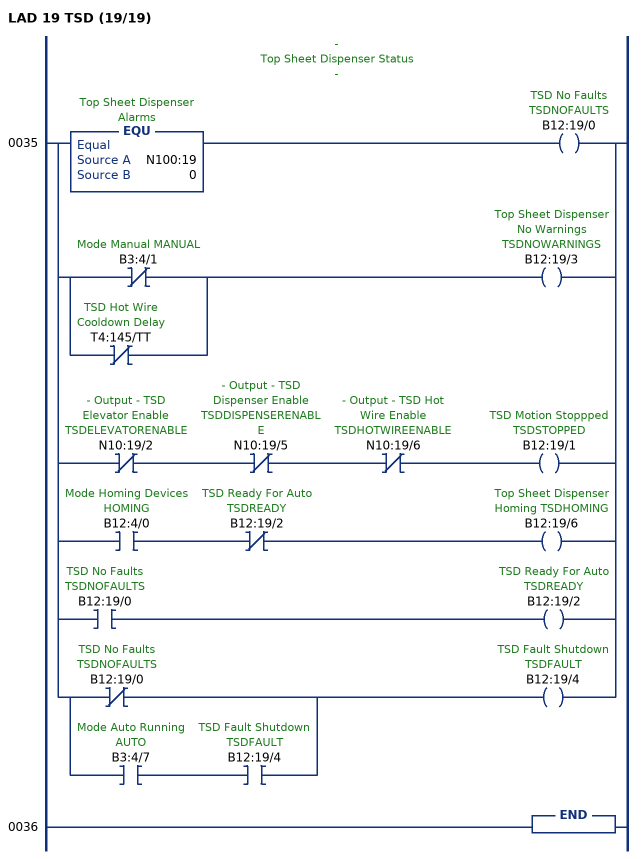
% Rung: 35 %
% -
% 
% Top Sheet Dispenser Status
% 
% - %
SOR BST EQU N100:19 0 OTE B12:19/0 NXB BST XIO B3:4/1 NXB XIO T4:145/TT BND OTE B12:19/3 NXB XIO N10:19/2 XIO N10:19/5 XIO N10:19/6 OTE B12:19/1 NXB XIC B12:4/0 XIO B12:19/2 OTE B12:19/6 NXB XIC B12:19/0 OTE B12:19/2 NXB BST XIO B12:19/0 NXB XIC B3:4/7 XIC B12:19/4 BND OTE B12:19/4 BND EOR
%   N100:19  "Top Sheet Dispenser Alarms" %
%   B12:19/0  TSDNOFAULTS  "TSD No Faults" %
%   B3:4/1  MANUAL  "Mode Manual" %
%   T4:145  "TSD Hot Wire Cooldown Delay" %
%   B12:19/3  TSDNOWARNINGS  "Top Sheet Dispenser No Warnings" %
%   N10:19/2  TSDELEVATORENABLE  "- Output - TSD Elevator Enable" %
%   N10:19/5  TSDDISPENSERENABLE  "- Output - TSD Dispenser Enable" %
%   N10:19/6  TSDHOTWIREENABLE  "- Output - TSD Hot Wire Enable" %
%   B12:19/1  TSDSTOPPED  "TSD Motion Stoppped" %
%   B12:4/0  HOMING  "Mode Homing Devices" %
%   B12:19/2  TSDREADY  "TSD Ready For Auto" %
%   B12:19/6  TSDHOMING  "Top Sheet Dispenser Homing" %
%   B3:4/7  AUTO  "Mode Auto Running" %
%   B12:19/4  TSDFAULT  "TSD Fault Shutdown" %
% Rung: 36 %
SOR END EOR

LADDER 27 "CONV IN 3"
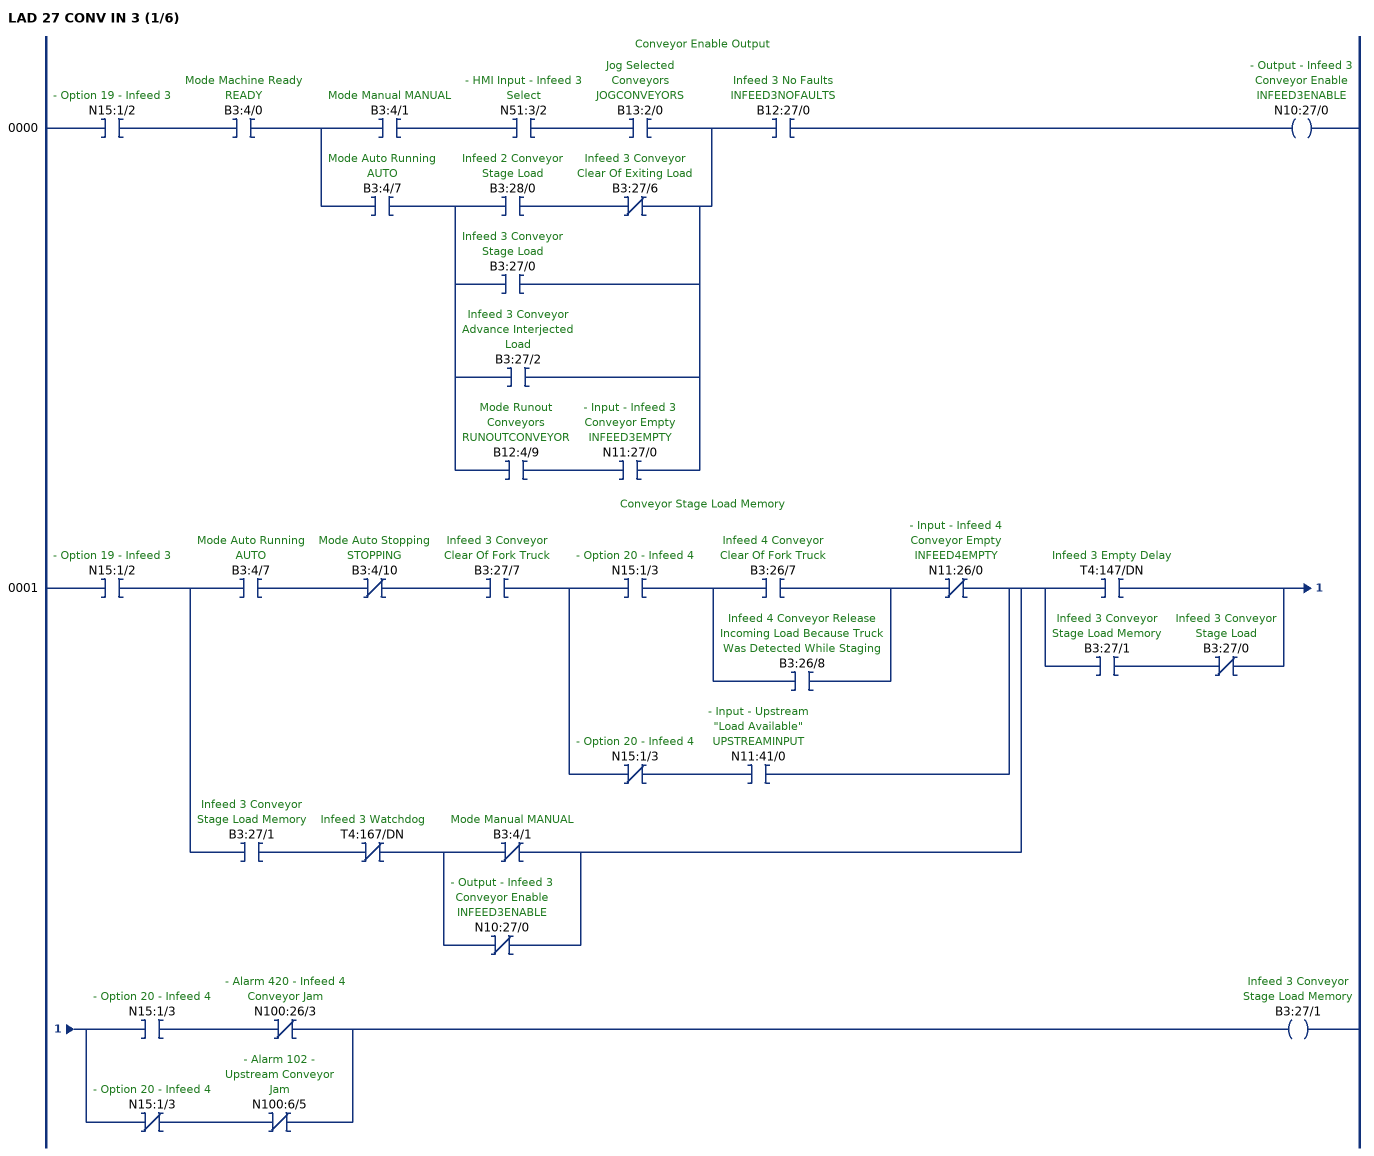
% Rung: 0 %
% Conveyor Enable Output %
SOR XIC N15:1/2 XIC B3:4/0 BST XIC B3:4/1 XIC N51:3/2 XIC B13:2/0 NXB XIC B3:4/7 BST XIC B3:28/0 XIO B3:27/6 NXB XIC B3:27/0 NXB XIC B3:27/2 NXB XIC B12:4/9 XIC N11:27/0 BND BND XIC B12:27/0 OTE N10:27/0 EOR
%   N15:1/2  "- Option 19 - Infeed 3" %
%   B3:4/0  READY  "Mode Machine Ready" %
%   B3:4/1  MANUAL  "Mode Manual" %
%   N51:3/2  "- HMI Input - Infeed 3 Select" %
%   B13:2/0  JOGCONVEYORS  "Jog Selected Conveyors" %
%   B3:4/7  AUTO  "Mode Auto Running" %
%   B3:28/0  "Infeed 2 Conveyor Stage Load" %
%   B3:27/6  "Infeed 3 Conveyor Clear Of Exiting Load" %
%   B3:27/0  "Infeed 3 Conveyor Stage Load" %
%   B3:27/2  "Infeed 3 Conveyor Advance Interjected Load" %
%   B12:4/9  RUNOUTCONVEYOR  "Mode Runout Conveyors" %
%   N11:27/0  INFEED3EMPTY  "- Input - Infeed 3 Conveyor Empty" %
%   B12:27/0  INFEED3NOFAULTS  "Infeed 3 No Faults" %
%   N10:27/0  INFEED3ENABLE  "- Output - Infeed 3 Conveyor Enable" %
% Rung: 1 %
% Conveyor Stage Load Memory %
SOR XIC N15:1/2 BST XIC B3:4/7 XIO B3:4/10 XIC B3:27/7 BST XIC N15:1/3 BST XIC B3:26/7 NXB XIC B3:26/8 BND XIO N11:26/0 NXB XIO N15:1/3 XIC N11:41/0 BND NXB XIC B3:27/1 XIO T4:167/DN BST XIO B3:4/1 NXB XIO N10:27/0 BND BND BST XIC T4:147/DN NXB XIC B3:27/1 XIO B3:27/0 BND BST XIC N15:1/3 XIO N100:26/3 NXB XIO N15:1/3 XIO N100:6/5 BND OTE B3:27/1 EOR
%   N15:1/2  "- Option 19 - Infeed 3" %
%   B3:4/7  AUTO  "Mode Auto Running" %
%   B3:4/10  STOPPING  "Mode Auto Stopping" %
%   B3:27/7  "Infeed 3 Conveyor Clear Of Fork Truck" %
%   N15:1/3  "- Option 20 - Infeed 4" %
%   B3:26/7  "Infeed 4 Conveyor Clear Of Fork Truck" %
%   B3:26/8  "Infeed 4 Conveyor Release Incoming Load Because Truck Was Detected While Staging" %
%   N11:26/0  INFEED4EMPTY  "- Input - Infeed 4 Conveyor Empty" %
%   N11:41/0  UPSTREAMINPUT  "- Input - Upstream "Load Available"" %
%   B3:27/1  "Infeed 3 Conveyor Stage Load Memory" %
%   T4:167  "Infeed 3 Watchdog" %
%   B3:4/1  MANUAL  "Mode Manual" %
%   N10:27/0  INFEED3ENABLE  "- Output - Infeed 3 Conveyor Enable" %
%   T4:147  "Infeed 3 Empty Delay" %
%   B3:27/0  "Infeed 3 Conveyor Stage Load" %
%   N100:26/3  "- Alarm 420 - Infeed 4 Conveyor Jam" %
%   N100:6/5  "- Alarm 102 - Upstream Conveyor Jam" %

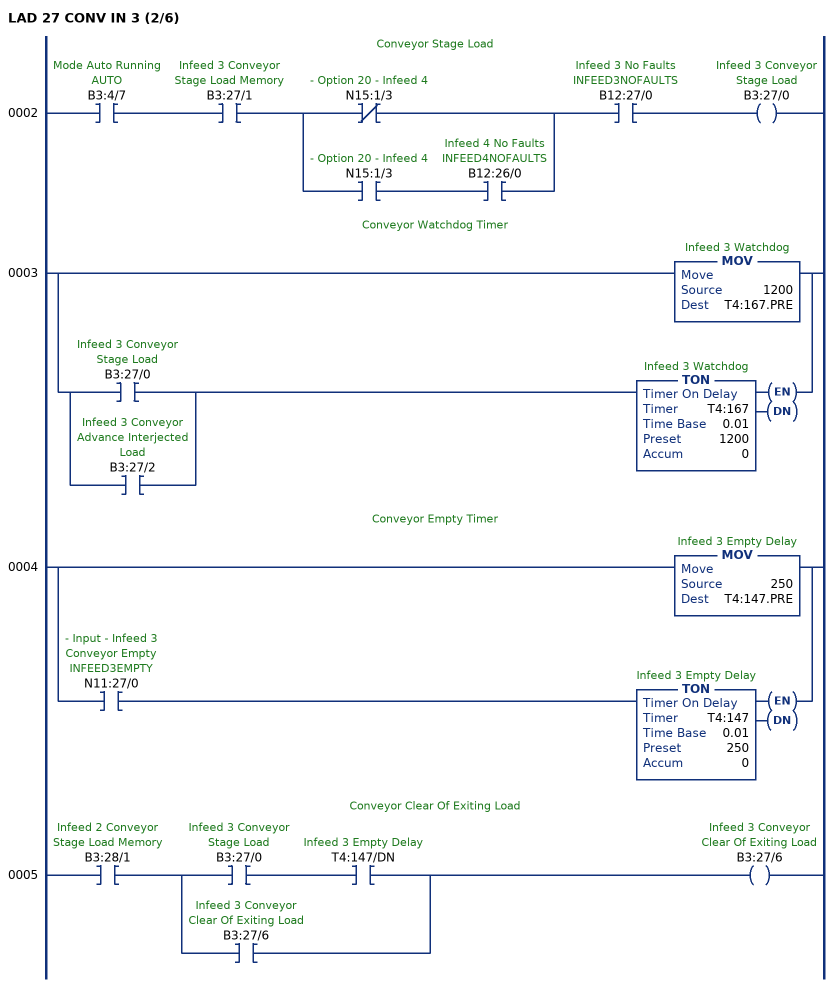
% Rung: 2 %
% Conveyor Stage Load %
SOR XIC B3:4/7 XIC B3:27/1 BST XIO N15:1/3 NXB XIC N15:1/3 XIC B12:26/0 BND XIC B12:27/0 OTE B3:27/0 EOR
%   B3:4/7  AUTO  "Mode Auto Running" %
%   B3:27/1  "Infeed 3 Conveyor Stage Load Memory" %
%   N15:1/3  "- Option 20 - Infeed 4" %
%   B12:26/0  INFEED4NOFAULTS  "Infeed 4 No Faults" %
%   B12:27/0  INFEED3NOFAULTS  "Infeed 3 No Faults" %
%   B3:27/0  "Infeed 3 Conveyor Stage Load" %
% Rung: 3 %
% Conveyor Watchdog Timer %
SOR BST MOV 1200 T4:167.PRE NXB BST XIC B3:27/0 NXB XIC B3:27/2 BND TON T4:167 0.01 1200 0 BND EOR
%   T4:167  "Infeed 3 Watchdog" %
%   B3:27/0  "Infeed 3 Conveyor Stage Load" %
%   B3:27/2  "Infeed 3 Conveyor Advance Interjected Load" %
% Rung: 4 %
% Conveyor Empty Timer %
SOR BST MOV 250 T4:147.PRE NXB XIC N11:27/0 TON T4:147 0.01 250 0 BND EOR
%   T4:147  "Infeed 3 Empty Delay" %
%   N11:27/0  INFEED3EMPTY  "- Input - Infeed 3 Conveyor Empty" %
% Rung: 5 %
% Conveyor Clear Of Exiting Load %
SOR XIC B3:28/1 BST XIC B3:27/0 XIC T4:147/DN NXB XIC B3:27/6 BND OTE B3:27/6 EOR
%   B3:28/1  "Infeed 2 Conveyor Stage Load Memory" %
%   B3:27/0  "Infeed 3 Conveyor Stage Load" %
%   T4:147  "Infeed 3 Empty Delay" %
%   B3:27/6  "Infeed 3 Conveyor Clear Of Exiting Load" %

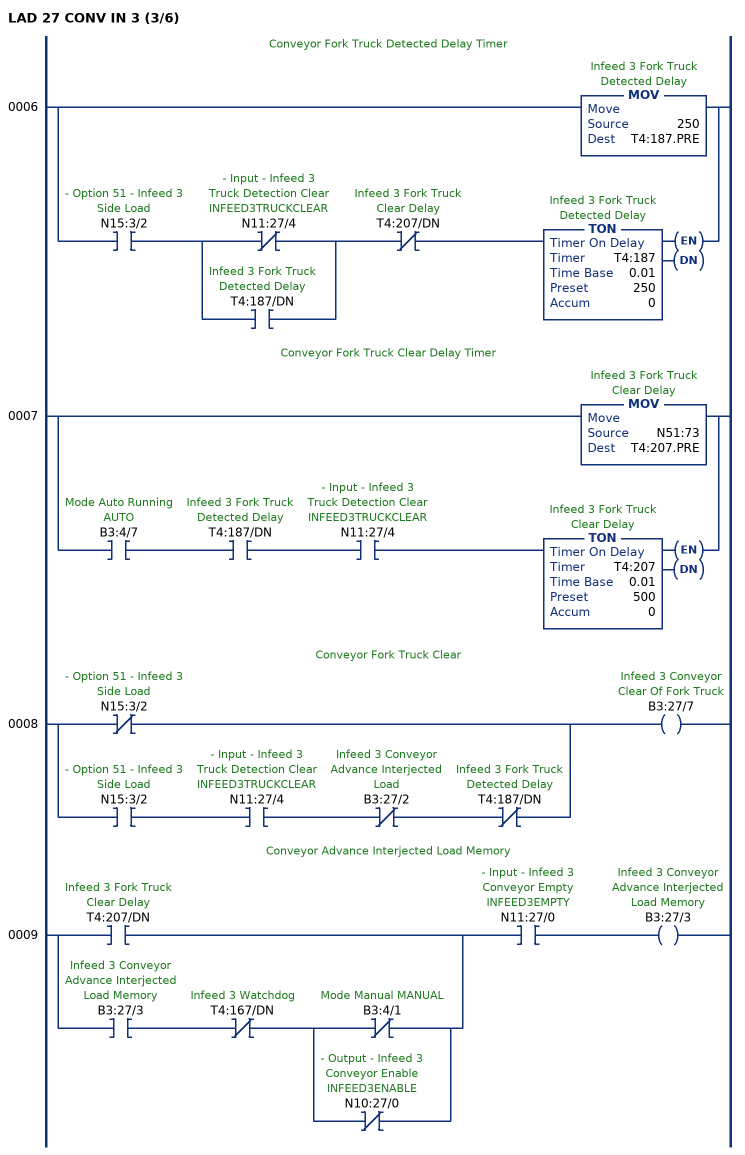
% Rung: 6 %
% Conveyor Fork Truck Detected Delay Timer %
SOR BST MOV 250 T4:187.PRE NXB XIC N15:3/2 BST XIO N11:27/4 NXB XIC T4:187/DN BND XIO T4:207/DN TON T4:187 0.01 250 0 BND EOR
%   T4:187  "Infeed 3 Fork Truck Detected Delay" %
%   N15:3/2  "- Option 51 - Infeed 3 Side Load" %
%   N11:27/4  INFEED3TRUCKCLEAR  "- Input - Infeed 3 Truck Detection Clear" %
%   T4:207  "Infeed 3 Fork Truck Clear Delay" %
% Rung: 7 %
% Conveyor Fork Truck Clear Delay Timer %
SOR BST MOV N51:73 T4:207.PRE NXB XIC B3:4/7 XIC T4:187/DN XIC N11:27/4 TON T4:207 0.01 500 0 BND EOR
%   N51:73  "- HMI Input - Preset Truck Clear" %
%   T4:207  "Infeed 3 Fork Truck Clear Delay" %
%   B3:4/7  AUTO  "Mode Auto Running" %
%   T4:187  "Infeed 3 Fork Truck Detected Delay" %
%   N11:27/4  INFEED3TRUCKCLEAR  "- Input - Infeed 3 Truck Detection Clear" %
% Rung: 8 %
% Conveyor Fork Truck Clear %
SOR BST XIO N15:3/2 NXB XIC N15:3/2 XIC N11:27/4 XIO B3:27/2 XIO T4:187/DN BND OTE B3:27/7 EOR
%   N15:3/2  "- Option 51 - Infeed 3 Side Load" %
%   N11:27/4  INFEED3TRUCKCLEAR  "- Input - Infeed 3 Truck Detection Clear" %
%   B3:27/2  "Infeed 3 Conveyor Advance Interjected Load" %
%   T4:187  "Infeed 3 Fork Truck Detected Delay" %
%   B3:27/7  "Infeed 3 Conveyor Clear Of Fork Truck" %
% Rung: 9 %
% Conveyor Advance Interjected Load Memory %
SOR BST XIC T4:207/DN NXB XIC B3:27/3 XIO T4:167/DN BST XIO B3:4/1 NXB XIO N10:27/0 BND BND XIC N11:27/0 OTE B3:27/3 EOR
%   T4:207  "Infeed 3 Fork Truck Clear Delay" %
%   B3:27/3  "Infeed 3 Conveyor Advance Interjected Load Memory" %
%   T4:167  "Infeed 3 Watchdog" %
%   B3:4/1  MANUAL  "Mode Manual" %
%   N10:27/0  INFEED3ENABLE  "- Output - Infeed 3 Conveyor Enable" %
%   N11:27/0  INFEED3EMPTY  "- Input - Infeed 3 Conveyor Empty" %

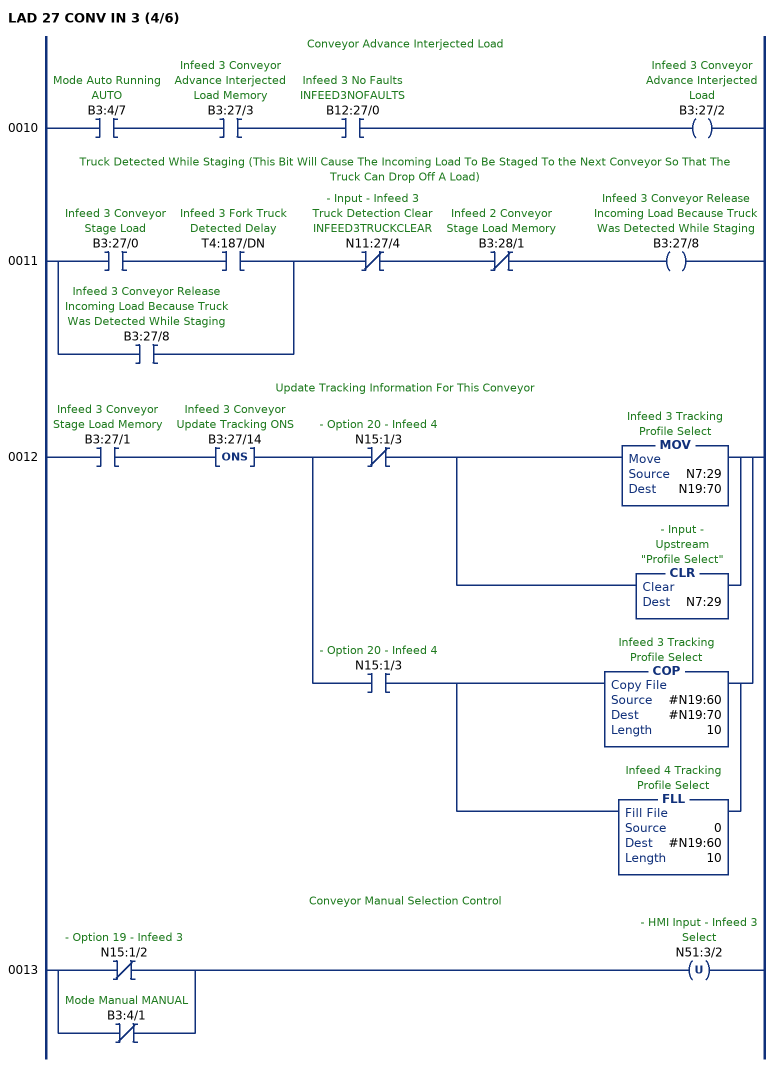
% Rung: 10 %
% Conveyor Advance Interjected Load %
SOR XIC B3:4/7 XIC B3:27/3 XIC B12:27/0 OTE B3:27/2 EOR
%   B3:4/7  AUTO  "Mode Auto Running" %
%   B3:27/3  "Infeed 3 Conveyor Advance Interjected Load Memory" %
%   B12:27/0  INFEED3NOFAULTS  "Infeed 3 No Faults" %
%   B3:27/2  "Infeed 3 Conveyor Advance Interjected Load" %
% Rung: 11 %
% Truck Detected While Staging (This Bit Will Cause The Incoming Load To Be Staged To the Next Conveyor So That The Truck Can Drop Off A Load) %
SOR BST XIC B3:27/0 XIC T4:187/DN NXB XIC B3:27/8 BND XIO N11:27/4 XIO B3:28/1 OTE B3:27/8 EOR
%   B3:27/0  "Infeed 3 Conveyor Stage Load" %
%   T4:187  "Infeed 3 Fork Truck Detected Delay" %
%   B3:27/8  "Infeed 3 Conveyor Release Incoming Load Because Truck Was Detected While Staging" %
%   N11:27/4  INFEED3TRUCKCLEAR  "- Input - Infeed 3 Truck Detection Clear" %
%   B3:28/1  "Infeed 2 Conveyor Stage Load Memory" %
% Rung: 12 %
% Update Tracking Information For This Conveyor %
SOR XIC B3:27/1 ONS B3:27/14 BST XIO N15:1/3 BST MOV N7:29 N19:70 NXB CLR N7:29 BND NXB XIC N15:1/3 BST COP #N19:60 #N19:70 10 NXB FLL 0 #N19:60 10 BND BND EOR
%   B3:27/1  "Infeed 3 Conveyor Stage Load Memory" %
%   B3:27/14  "Infeed 3 Conveyor Update Tracking ONS" %
%   N15:1/3  "- Option 20 - Infeed 4" %
%   N7:29  "- Input - Upstream "Profile Select"" %
%   N19:70  "Infeed 3 Tracking Profile Select" %
%   N19:60  "Infeed 4 Tracking Profile Select" %
% Rung: 13 %
% Conveyor Manual Selection Control %
SOR BST XIO N15:1/2 NXB XIO B3:4/1 BND OTU N51:3/2 EOR
%   N15:1/2  "- Option 19 - Infeed 3" %
%   B3:4/1  MANUAL  "Mode Manual" %
%   N51:3/2  "- HMI Input - Infeed 3 Select" %

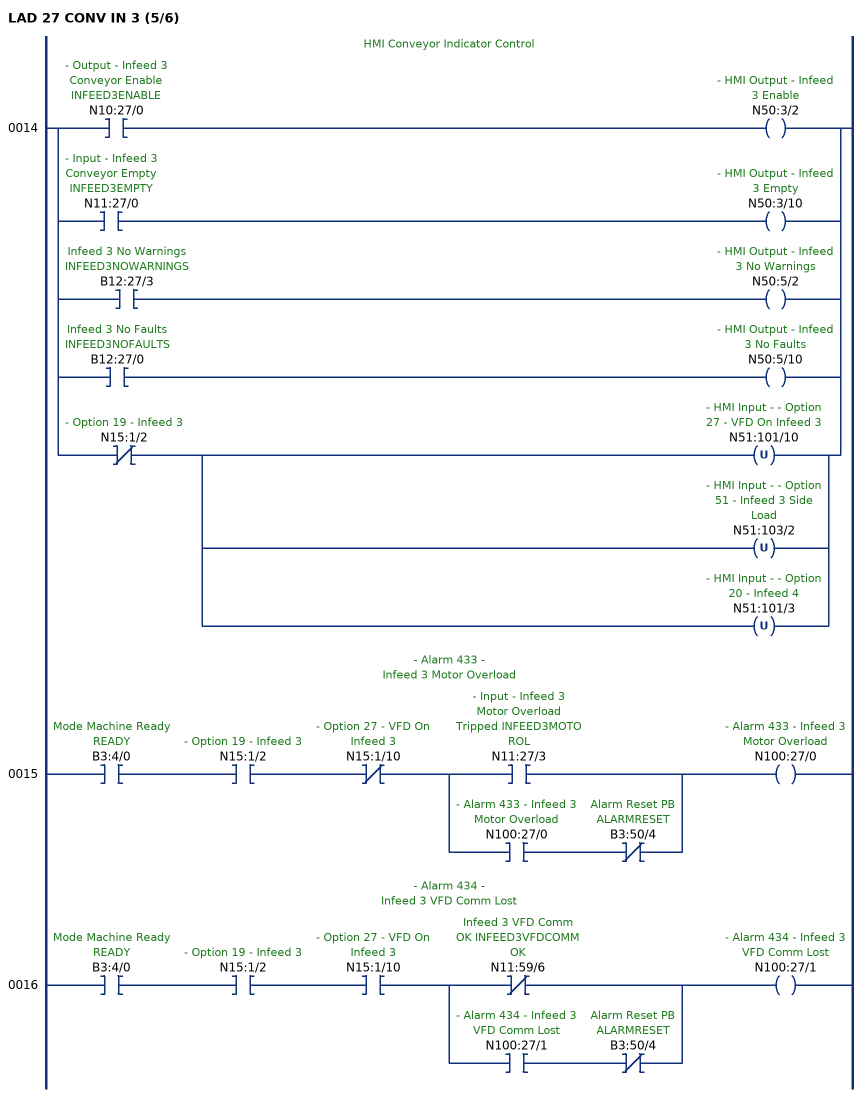
% Rung: 14 %
% HMI Conveyor Indicator Control %
SOR BST XIC N10:27/0 OTE N50:3/2 NXB XIC N11:27/0 OTE N50:3/10 NXB XIC B12:27/3 OTE N50:5/2 NXB XIC B12:27/0 OTE N50:5/10 NXB XIO N15:1/2 BST OTU N51:101/10 NXB OTU N51:103/2 NXB OTU N51:101/3 BND BND EOR
%   N10:27/0  INFEED3ENABLE  "- Output - Infeed 3 Conveyor Enable" %
%   N50:3/2  "- HMI Output - Infeed 3 Enable" %
%   N11:27/0  INFEED3EMPTY  "- Input - Infeed 3 Conveyor Empty" %
%   N50:3/10  "- HMI Output - Infeed 3 Empty" %
%   B12:27/3  INFEED3NOWARNINGS  "Infeed 3 No Warnings" %
%   N50:5/2  "- HMI Output - Infeed 3 No Warnings" %
%   B12:27/0  INFEED3NOFAULTS  "Infeed 3 No Faults" %
%   N50:5/10  "- HMI Output - Infeed 3 No Faults" %
%   N15:1/2  "- Option 19 - Infeed 3" %
%   N51:101/10  "- HMI Input - - Option 27 - VFD On Infeed 3" %
%   N51:103/2  "- HMI Input - - Option 51 - Infeed 3 Side Load" %
%   N51:101/3  "- HMI Input - - Option 20 - Infeed 4" %
% Rung: 15 %
% - Alarm 433 -
% 
% Infeed 3 Motor Overload %
SOR XIC B3:4/0 XIC N15:1/2 XIO N15:1/10 BST XIC N11:27/3 NXB XIC N100:27/0 XIO B3:50/4 BND OTE N100:27/0 EOR
%   B3:4/0  READY  "Mode Machine Ready" %
%   N15:1/2  "- Option 19 - Infeed 3" %
%   N15:1/10  "- Option 27 - VFD On Infeed 3" %
%   N11:27/3  INFEED3MOTOROL  "- Input - Infeed 3 Motor Overload Tripped" %
%   N100:27/0  "- Alarm 433 - Infeed 3 Motor Overload" %
%   B3:50/4  ALARMRESET  "Alarm Reset PB" %
% Rung: 16 %
% - Alarm 434 -
% 
% Infeed 3 VFD Comm Lost %
SOR XIC B3:4/0 XIC N15:1/2 XIC N15:1/10 BST XIO N11:59/6 NXB XIC N100:27/1 XIO B3:50/4 BND OTE N100:27/1 EOR
%   B3:4/0  READY  "Mode Machine Ready" %
%   N15:1/2  "- Option 19 - Infeed 3" %
%   N15:1/10  "- Option 27 - VFD On Infeed 3" %
%   N11:59/6  INFEED3VFDCOMMOK  "Infeed 3 VFD Comm OK" %
%   N100:27/1  "- Alarm 434 - Infeed 3 VFD Comm Lost" %
%   B3:50/4  ALARMRESET  "Alarm Reset PB" %

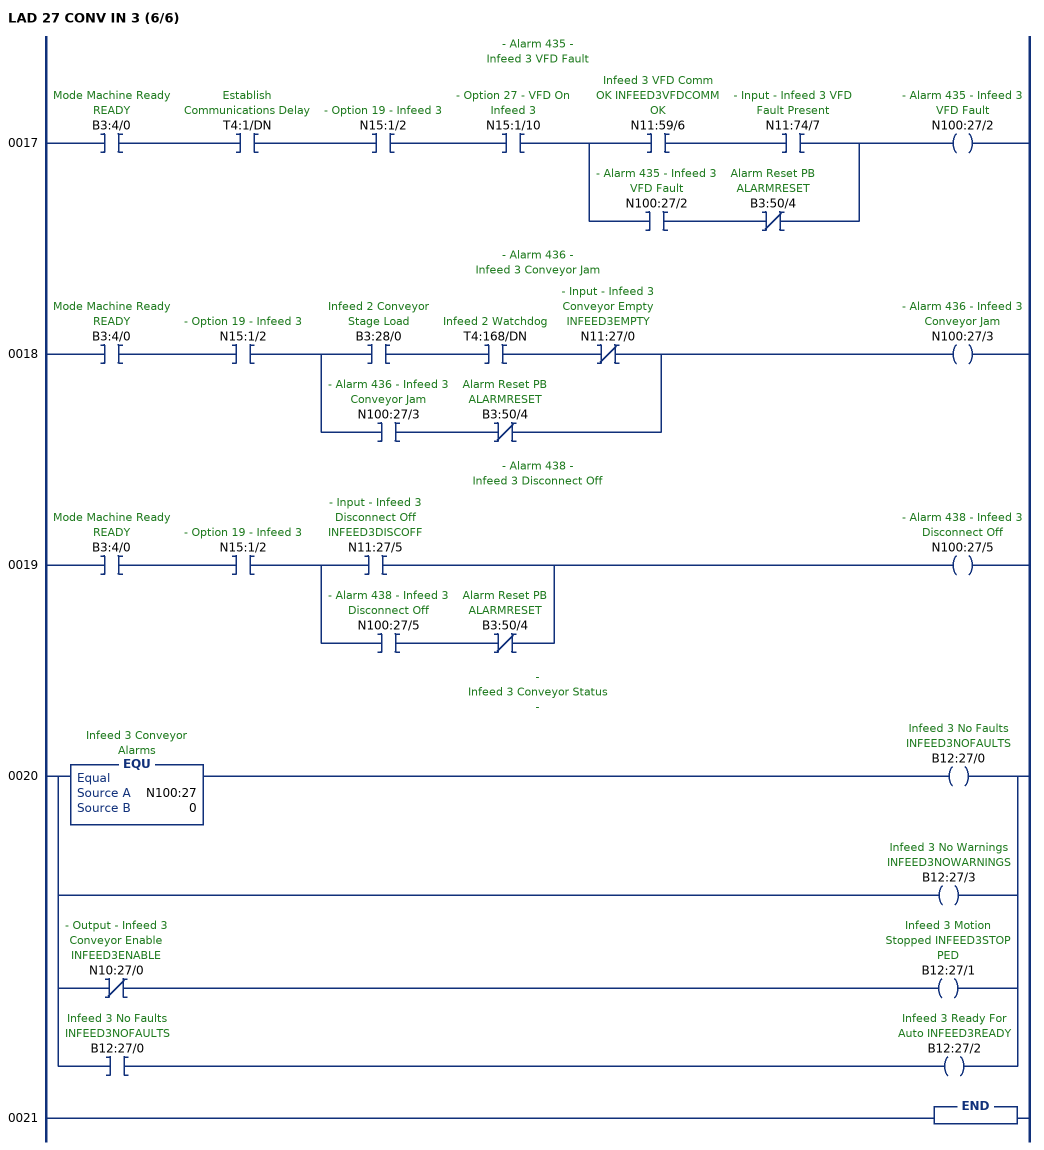
% Rung: 17 %
% - Alarm 435 -
% 
% Infeed 3 VFD Fault %
SOR XIC B3:4/0 XIC T4:1/DN XIC N15:1/2 XIC N15:1/10 BST XIC N11:59/6 XIC N11:74/7 NXB XIC N100:27/2 XIO B3:50/4 BND OTE N100:27/2 EOR
%   B3:4/0  READY  "Mode Machine Ready" %
%   T4:1  "Establish Communications Delay" %
%   N15:1/2  "- Option 19 - Infeed 3" %
%   N15:1/10  "- Option 27 - VFD On Infeed 3" %
%   N11:59/6  INFEED3VFDCOMMOK  "Infeed 3 VFD Comm OK" %
%   N11:74/7  "- Input - Infeed 3 VFD Fault Present" %
%   N100:27/2  "- Alarm 435 - Infeed 3 VFD Fault" %
%   B3:50/4  ALARMRESET  "Alarm Reset PB" %
% Rung: 18 %
% - Alarm 436 -
% 
% Infeed 3 Conveyor Jam %
SOR XIC B3:4/0 XIC N15:1/2 BST XIC B3:28/0 XIC T4:168/DN XIO N11:27/0 NXB XIC N100:27/3 XIO B3:50/4 BND OTE N100:27/3 EOR
%   B3:4/0  READY  "Mode Machine Ready" %
%   N15:1/2  "- Option 19 - Infeed 3" %
%   B3:28/0  "Infeed 2 Conveyor Stage Load" %
%   T4:168  "Infeed 2 Watchdog" %
%   N11:27/0  INFEED3EMPTY  "- Input - Infeed 3 Conveyor Empty" %
%   N100:27/3  "- Alarm 436 - Infeed 3 Conveyor Jam" %
%   B3:50/4  ALARMRESET  "Alarm Reset PB" %
% Rung: 19 %
% - Alarm 438 -
% 
% Infeed 3 Disconnect Off %
SOR XIC B3:4/0 XIC N15:1/2 BST XIC N11:27/5 NXB XIC N100:27/5 XIO B3:50/4 BND OTE N100:27/5 EOR
%   B3:4/0  READY  "Mode Machine Ready" %
%   N15:1/2  "- Option 19 - Infeed 3" %
%   N11:27/5  INFEED3DISCOFF  "- Input - Infeed 3 Disconnect Off" %
%   N100:27/5  "- Alarm 438 - Infeed 3 Disconnect Off" %
%   B3:50/4  ALARMRESET  "Alarm Reset PB" %
% Rung: 20 %
% -
% 
% Infeed 3 Conveyor Status
% 
% - %
SOR BST EQU N100:27 0 OTE B12:27/0 NXB OTE B12:27/3 NXB XIO N10:27/0 OTE B12:27/1 NXB XIC B12:27/0 OTE B12:27/2 BND EOR
%   N100:27  "Infeed 3 Conveyor Alarms" %
%   B12:27/0  INFEED3NOFAULTS  "Infeed 3 No Faults" %
%   B12:27/3  INFEED3NOWARNINGS  "Infeed 3 No Warnings" %
%   N10:27/0  INFEED3ENABLE  "- Output - Infeed 3 Conveyor Enable" %
%   B12:27/1  INFEED3STOPPED  "Infeed 3 Motion Stopped" %
%   B12:27/2  INFEED3READY  "Infeed 3 Ready For Auto" %
% Rung: 21 %
SOR END EOR

LADDER 28 "CONV IN 2"
